C07141=1012.979,-24.500,-114.900,-28.755,51.503,-32.003
C07142=1012.980,-24.266,-114.919,-28.753,51.485,-32.004
C07143=1012.980,-24.032,-114.938,-28.751,51.466,-32.006
C07144=1012.980,-23.797,-114.958,-28.749,51.447,-32.007
C07145=1012.981,-23.564,-114.978,-28.747,51.429,-32.008
C07146=1012.981,-23.329,-114.997,-28.745,51.412,-32.007
C07147=1012.981,-23.095,-115.017,-28.743,51.394,-32.009
C07148=1012.982,-22.861,-115.036,-28.741,51.376,-32.010
C07149=1012.982,-22.628,-115.056,-28.739,51.359,-32.010
C07150=1012.982,-22.394,-115.076,-28.737,51.342,-32.011
C07151=1012.982,-22.159,-115.095,-28.736,51.326,-32.012
C07152=1012.983,-21.925,-115.114,-28.734,51.309,-32.012
C07153=1012.983,-21.691,-115.135,-28.732,51.292,-32.013
C07154=1012.983,-21.457,-115.154,-28.730,51.276,-32.014
C07155=1012.984,-21.223,-115.173,-28.728,51.261,-32.015
C07156=1012.983,-20.989,-115.193,-28.726,51.246,-32.014
C07157=1012.984,-20.755,-115.213,-28.725,51.230,-32.015
C07158=1012.985,-20.521,-115.232,-28.723,51.215,-32.015
C07159=1012.984,-20.243,-115.255,-28.721,51.197,-32.016
C07160=1012.985,-19.894,-115.285,-28.718,51.175,-32.016
C07161=1012.986,-19.633,-115.306,-28.717,51.160,-32.017
C07162=1012.986,-19.334,-115.331,-28.714,51.142,-32.017
C07163=1012.986,-19.008,-115.359,-28.712,51.123,-32.017
C07164=1012.987,-18.676,-115.386,-28.710,51.105,-32.018
C07165=1012.986,-18.359,-115.413,-28.708,51.087,-32.018
C07166=1012.987,-18.074,-115.437,-28.706,51.072,-32.017
C07167=1012.987,-17.827,-115.458,-28.704,51.058,-32.018
C07168=1012.987,-17.596,-115.477,-28.703,51.046,-32.018
C07169=1012.987,-17.366,-115.497,-28.702,51.035,-32.017
C07170=1012.988,-17.131,-115.516,-28.700,51.023,-32.017
C07171=1012.988,-16.894,-115.536,-28.699,51.011,-32.017
C07172=1012.987,-16.657,-115.556,-28.697,50.999,-32.017
C07173=1012.988,-16.421,-115.575,-28.696,50.989,-32.016
C07174=1012.988,-16.187,-115.595,-28.695,50.979,-32.016
C07175=1012.988,-15.950,-115.616,-28.693,50.967,-32.017
C07176=1012.989,-15.715,-115.634,-28.692,50.957,-32.016
C07177=1012.988,-15.481,-115.655,-28.691,50.947,-32.016
C07178=1012.989,-15.253,-115.673,-28.690,50.937,-32.016
C07179=1012.989,-15.025,-115.692,-28.688,50.928,-32.014
C07180=1012.989,-14.801,-115.712,-28.687,50.919,-32.013
C07181=1012.988,-14.578,-115.730,-28.686,50.909,-32.013
C07182=1012.989,-14.355,-115.749,-28.685,50.901,-32.012
C07183=1012.989,-14.131,-115.768,-28.683,50.893,-32.011
C07184=1012.989,-13.906,-115.786,-28.682,50.885,-32.009
C07185=1012.989,-13.676,-115.806,-28.681,50.878,-32.009
C07186=1012.989,-13.443,-115.825,-28.680,50.869,-32.008
C07187=1012.989,-13.206,-115.845,-28.679,50.861,-32.007
C07188=1012.989,-12.965,-115.865,-28.678,50.853,-32.007
C07189=1012.989,-12.720,-115.886,-28.677,50.846,-32.007
C07190=1012.990,-12.475,-115.906,-28.676,50.838,-32.006
C07191=1012.990,-12.228,-115.927,-28.675,50.831,-32.004
C07192=1012.989,-11.982,-115.948,-28.674,50.824,-32.003
C07193=1012.989,-11.734,-115.968,-28.673,50.817,-32.003
C07194=1012.989,-11.486,-115.990,-28.672,50.810,-32.001
C07195=1012.989,-11.237,-116.011,-28.671,50.804,-32.000
C07196=1012.989,-10.989,-116.031,-28.670,50.798,-31.999
C07197=1012.989,-10.739,-116.052,-28.669,50.793,-31.997
C07198=1012.989,-10.489,-116.073,-28.668,50.787,-31.996
C07199=1012.989,-10.239,-116.094,-28.667,50.782,-31.994
C07200=1012.990,-9.989,-116.115,-28.666,50.776,-31.993
C07201=1012.989,-9.738,-116.136,-28.666,50.772,-31.991
C07202=1012.989,-9.487,-116.157,-28.665,50.767,-31.989
C07203=1012.989,-9.236,-116.179,-28.664,50.763,-31.988
C07204=1012.989,-8.985,-116.199,-28.663,50.758,-31.986
C07205=1012.989,-8.733,-116.221,-28.662,50.754,-31.985
C07206=1012.989,-8.481,-116.242,-28.661,50.751,-31.982
C07207=1012.989,-8.230,-116.263,-28.661,50.748,-31.981
C07208=1012.989,-7.978,-116.284,-28.660,50.745,-31.979
C07209=1012.989,-7.724,-116.305,-28.659,50.742,-31.976
C07210=1012.989,-7.470,-116.327,-28.659,50.739,-31.975
C07211=1012.988,-7.215,-116.348,-28.658,50.737,-31.974
C07212=1012.988,-6.959,-116.369,-28.658,50.735,-31.970
C07213=1012.988,-6.702,-116.391,-28.657,50.734,-31.969
C07214=1012.987,-6.444,-116.413,-28.657,50.731,-31.967
C07215=1012.988,-6.186,-116.434,-28.656,50.730,-31.964
C07216=1012.987,-5.928,-116.456,-28.655,50.729,-31.961
C07217=1012.987,-5.670,-116.477,-28.655,50.728,-31.960
C07218=1012.987,-5.413,-116.499,-28.655,50.728,-31.957
C07219=1012.986,-5.161,-116.521,-28.654,50.728,-31.955
C07220=1012.987,-4.917,-116.541,-28.654,50.728,-31.953
C07221=1012.987,-4.682,-116.561,-28.654,50.728,-31.951
C07222=1012.986,-4.453,-116.580,-28.653,50.729,-31.948
C07223=1012.986,-4.227,-116.599,-28.653,50.729,-31.946
C07224=1012.986,-4.001,-116.618,-28.652,50.731,-31.943
C07225=1012.986,-3.771,-116.637,-28.652,50.731,-31.939
C07226=1012.986,-3.534,-116.658,-28.652,50.732,-31.938
C07227=1012.985,-3.292,-116.678,-28.651,50.734,-31.935
C07228=1012.985,-3.047,-116.698,-28.651,50.736,-31.933
C07229=1012.985,-2.802,-116.719,-28.651,50.738,-31.931
C07230=1012.985,-2.558,-116.739,-28.651,50.741,-31.926
C07231=1012.984,-2.315,-116.760,-28.651,50.743,-31.924
C07232=1012.984,-2.072,-116.781,-28.651,50.746,-31.922
C07233=1012.984,-1.830,-116.800,-28.650,50.749,-31.919
C07234=1012.983,-1.589,-116.821,-28.650,50.753,-31.915
C07235=1012.983,-1.348,-116.841,-28.650,50.755,-31.913
C07236=1012.983,-1.109,-116.861,-28.650,50.758,-31.910
C07237=1012.982,-0.869,-116.882,-28.650,50.763,-31.907
C07238=1012.983,-0.631,-116.902,-28.650,50.767,-31.905
C07239=1012.982,-0.393,-116.922,-28.650,50.772,-31.901
C07240=1012.982,-0.156,-116.941,-28.650,50.776,-31.898
C07241=1012.982,0.079,-116.961,-28.650,50.780,-31.895
C07242=1012.980,0.314,-116.981,-28.650,50.785,-31.891
C07243=1012.980,0.548,-117.001,-28.650,50.790,-31.889
C07244=1012.980,0.784,-117.021,-28.650,50.795,-31.885
C07245=1012.980,1.019,-117.040,-28.650,50.801,-31.882
C07246=1012.980,1.256,-117.060,-28.650,50.807,-31.878
C07247=1012.979,1.492,-117.080,-28.650,50.813,-31.875
C07248=1012.979,1.727,-117.100,-28.650,50.819,-31.872
C07249=1012.978,1.956,-117.119,-28.651,50.825,-31.868
C07250=1012.978,2.177,-117.138,-28.651,50.832,-31.866
C07251=1012.978,2.585,-117.172,-28.651,50.843,-31.859
C07252=1012.977,2.969,-117.205,-28.652,50.856,-31.853
C07253=1012.976,3.360,-117.238,-28.652,50.868,-31.847
C07254=1012.975,3.569,-117.255,-28.652,50.875,-31.844
C07255=1012.976,3.788,-117.273,-28.653,50.883,-31.840
C07256=1012.975,4.016,-117.293,-28.653,50.890,-31.836
C07257=1012.974,4.249,-117.312,-28.653,50.899,-31.833
C07258=1012.974,4.481,-117.332,-28.654,50.907,-31.829
C07259=1012.974,4.713,-117.351,-28.654,50.916,-31.825
C07260=1012.973,4.944,-117.371,-28.654,50.925,-31.822
C07261=1012.973,5.176,-117.390,-28.655,50.935,-31.818
C07262=1012.972,5.408,-117.410,-28.655,50.943,-31.814
C07263=1012.972,5.641,-117.430,-28.656,50.953,-31.810
C07264=1012.971,5.875,-117.449,-28.656,50.963,-31.806
C07265=1012.971,6.109,-117.469,-28.656,50.973,-31.802
C07266=1012.970,6.343,-117.488,-28.657,50.983,-31.798
C07267=1012.970,6.576,-117.509,-28.657,50.993,-31.794
C07268=1012.970,6.806,-117.528,-28.658,51.004,-31.789
C07269=1012.969,7.036,-117.547,-28.658,51.015,-31.786
C07270=1012.968,7.263,-117.566,-28.659,51.025,-31.782
C07271=1012.968,7.489,-117.585,-28.660,51.037,-31.777
C07272=1012.967,7.715,-117.604,-28.660,51.048,-31.774
C07273=1012.966,7.939,-117.623,-28.661,51.059,-31.769
C07274=1012.966,8.162,-117.642,-28.661,51.070,-31.765
C07275=1012.965,8.385,-117.661,-28.662,51.082,-31.761
C07276=1012.965,8.608,-117.680,-28.662,51.093,-31.756
C07277=1012.965,8.830,-117.698,-28.663,51.106,-31.752
C07278=1012.964,9.052,-117.718,-28.664,51.118,-31.748
C07279=1012.964,9.275,-117.737,-28.664,51.130,-31.744
C07280=1012.963,9.498,-117.755,-28.665,51.142,-31.739
C07281=1012.962,9.721,-117.774,-28.666,51.154,-31.735
C07282=1012.962,9.944,-117.792,-28.667,51.167,-31.731
C07283=1012.961,10.168,-117.812,-28.667,51.180,-31.726
C07284=1012.961,10.394,-117.830,-28.668,51.194,-31.723
C07285=1012.960,10.618,-117.850,-28.669,51.207,-31.718
C07286=1012.960,10.839,-117.868,-28.670,51.222,-31.713
C07287=1012.959,11.056,-117.886,-28.670,51.234,-31.709
C07288=1012.958,11.272,-117.905,-28.671,51.248,-31.704
C07289=1012.958,11.488,-117.922,-28.672,51.262,-31.699
C07290=1012.957,11.708,-117.942,-28.673,51.276,-31.695
C07291=1012.956,11.931,-117.960,-28.673,51.290,-31.690
C07292=1012.956,12.158,-117.980,-28.674,51.305,-31.686
C07293=1012.955,12.387,-117.999,-28.675,51.320,-31.681
C07294=1012.954,12.615,-118.018,-28.676,51.336,-31.677
C07295=1012.954,12.844,-118.038,-28.677,51.351,-31.672
C07296=1012.954,13.072,-118.057,-28.678,51.367,-31.666
C07297=1012.953,13.300,-118.076,-28.679,51.383,-31.661
C07298=1012.952,13.527,-118.095,-28.680,51.399,-31.656
C07299=1012.952,13.755,-118.114,-28.681,51.416,-31.651
C07300=1012.951,13.982,-118.133,-28.682,51.432,-31.646
C07301=1012.951,14.208,-118.153,-28.683,51.449,-31.642
C07302=1012.949,14.434,-118.172,-28.684,51.465,-31.637
C07303=1012.949,14.660,-118.191,-28.685,51.481,-31.632
C07304=1012.948,14.886,-118.209,-28.686,51.499,-31.626
C07305=1012.948,15.113,-118.229,-28.687,51.516,-31.622
C07306=1012.947,15.340,-118.248,-28.688,51.534,-31.617
C07307=1012.946,15.565,-118.267,-28.689,51.552,-31.611
C07308=1012.945,15.792,-118.287,-28.690,51.570,-31.606
C07309=1012.944,16.019,-118.305,-28.691,51.588,-31.600
C07310=1012.944,16.247,-118.325,-28.693,51.606,-31.595
C07311=1012.943,16.474,-118.344,-28.694,51.625,-31.590
C07312=1012.943,16.703,-118.364,-28.695,51.643,-31.585
C07313=1012.942,16.931,-118.383,-28.696,51.663,-31.579
C07314=1012.940,17.161,-118.402,-28.697,51.682,-31.574
C07315=1012.940,17.392,-118.421,-28.699,51.702,-31.568
C07316=1012.939,17.623,-118.441,-28.700,51.722,-31.562
C07317=1012.939,17.855,-118.460,-28.701,51.742,-31.557
C07318=1012.938,18.087,-118.480,-28.702,51.762,-31.551
C07319=1012.937,18.320,-118.500,-28.704,51.783,-31.546
C07320=1012.936,18.553,-118.520,-28.705,51.803,-31.540
C07321=1012.935,18.786,-118.539,-28.707,51.824,-31.535
C07322=1012.934,19.048,-118.562,-28.708,51.848,-31.529
C07323=1012.933,19.353,-118.587,-28.710,51.876,-31.521
C07324=1012.931,19.749,-118.621,-28.712,51.913,-31.511
C07325=1012.930,20.049,-118.647,-28.714,51.941,-31.504
C07326=1012.929,20.367,-118.673,-28.716,51.972,-31.495
C07327=1012.928,20.687,-118.700,-28.718,52.002,-31.488
C07328=1012.927,20.997,-118.726,-28.720,52.033,-31.479
C07329=1012.926,21.286,-118.751,-28.722,52.062,-31.472
C07330=1012.925,21.545,-118.773,-28.724,52.088,-31.465
C07331=1012.923,21.956,-118.807,-28.726,52.129,-31.455
C07332=1012.922,22.369,-118.842,-28.729,52.172,-31.443
C07333=1012.921,22.713,-118.871,-28.731,52.208,-31.435
C07334=1012.919,23.005,-118.896,-28.733,52.238,-31.427
C07335=1012.918,23.306,-118.922,-28.736,52.270,-31.419
C07336=1012.917,23.669,-118.953,-28.738,52.309,-31.409
C07337=1012.916,23.879,-118.970,-28.740,52.331,-31.404
C07338=1012.916,24.101,-118.989,-28.741,52.356,-31.397
C07339=1012.914,24.333,-119.009,-28.743,52.381,-31.392
C07340=1012.913,24.569,-119.029,-28.745,52.408,-31.386
C07341=1012.912,24.804,-119.048,-28.746,52.434,-31.379
C07342=1012.911,25.040,-119.068,-28.748,52.460,-31.373
C07343=1012.910,25.276,-119.088,-28.750,52.486,-31.366
C07344=1012.909,25.512,-119.108,-28.752,52.514,-31.361
C07345=1012.907,25.749,-119.128,-28.754,52.542,-31.353
C07346=1012.907,25.986,-119.149,-28.756,52.568,-31.347
C07347=1012.906,26.222,-119.168,-28.757,52.596,-31.340
C07348=1012.905,26.459,-119.189,-28.759,52.624,-31.334
C07349=1012.904,26.694,-119.208,-28.761,52.651,-31.327
C07350=1012.903,26.929,-119.228,-28.763,52.680,-31.320
C07351=1012.902,27.163,-119.248,-28.765,52.708,-31.313
C07352=1012.901,27.396,-119.268,-28.767,52.737,-31.307
C07353=1012.899,27.630,-119.288,-28.769,52.764,-31.301
C07354=1012.899,27.864,-119.307,-28.770,52.794,-31.293
C07355=1012.898,28.099,-119.327,-28.772,52.822,-31.287
C07356=1012.897,28.333,-119.347,-28.774,52.851,-31.281
C07357=1012.896,28.566,-119.367,-28.777,52.881,-31.275
C07358=1012.895,28.802,-119.386,-28.778,52.910,-31.267
C07359=1012.893,29.037,-119.406,-28.780,52.939,-31.261
C07360=1012.892,29.272,-119.427,-28.782,52.969,-31.254
C07361=1012.891,29.507,-119.446,-28.784,53.000,-31.247
C07362=1012.890,29.744,-119.466,-28.786,53.030,-31.240
C07363=1012.889,29.978,-119.487,-28.789,53.061,-31.233
C07364=1012.888,30.214,-119.506,-28.790,53.091,-31.226
C07365=1012.887,30.449,-119.526,-28.793,53.122,-31.219
C07366=1012.886,30.684,-119.547,-28.795,53.153,-31.213
C07367=1012.885,30.919,-119.566,-28.797,53.184,-31.206
C07368=1012.883,31.155,-119.586,-28.799,53.217,-31.199
C07369=1012.882,31.390,-119.606,-28.801,53.248,-31.193
C07370=1012.882,31.624,-119.626,-28.804,53.281,-31.186
C07371=1012.881,31.860,-119.645,-28.806,53.312,-31.178
C07372=1012.879,32.095,-119.665,-28.808,53.344,-31.172
C07373=1012.878,32.330,-119.685,-28.810,53.377,-31.165
C07374=1012.877,32.565,-119.705,-28.812,53.409,-31.158
C07375=1012.876,32.801,-119.725,-28.815,53.442,-31.151
C07376=1012.874,33.036,-119.745,-28.817,53.475,-31.145
C07377=1012.874,33.272,-119.765,-28.819,53.509,-31.136
C07378=1012.873,33.507,-119.785,-28.821,53.542,-31.130
C07379=1012.871,33.742,-119.805,-28.824,53.577,-31.122
C07380=1012.870,33.978,-119.825,-28.826,53.609,-31.115
C07381=1012.869,34.213,-119.845,-28.828,53.644,-31.108
C07382=1012.868,34.448,-119.865,-28.831,53.678,-31.102
C07383=1012.866,34.684,-119.885,-28.833,53.712,-31.094
C07384=1012.865,34.919,-119.905,-28.835,53.747,-31.088
C07385=1012.864,35.154,-119.925,-28.838,53.782,-31.080
C07386=1012.862,35.389,-119.945,-28.840,53.817,-31.073
C07387=1012.861,35.625,-119.965,-28.843,53.852,-31.066
C07388=1012.860,35.860,-119.984,-28.845,53.888,-31.058
C07389=1012.859,36.095,-120.005,-28.847,53.923,-31.051
C07390=1012.857,36.330,-120.024,-28.850,53.958,-31.045
C07391=1012.856,36.566,-120.044,-28.852,53.995,-31.037
C07392=1012.855,36.801,-120.064,-28.855,54.032,-31.030
C07393=1012.854,37.036,-120.084,-28.857,54.067,-31.023
C07394=1012.853,37.271,-120.104,-28.860,54.103,-31.016
C07395=1012.851,37.507,-120.124,-28.862,54.140,-31.008
C07396=1012.850,37.742,-120.143,-28.865,54.177,-31.001
C07397=1012.848,37.978,-120.164,-28.868,54.215,-30.994
C07398=1012.847,38.214,-120.184,-28.870,54.251,-30.987
C07399=1012.846,38.449,-120.204,-28.873,54.289,-30.980
C07400=1012.845,38.684,-120.224,-28.875,54.327,-30.972
C07401=1012.844,38.919,-120.244,-28.878,54.364,-30.965
C07402=1012.843,39.155,-120.263,-28.880,54.403,-30.957
C07403=1012.841,39.390,-120.283,-28.883,54.440,-30.951
C07404=1012.840,39.626,-120.303,-28.886,54.479,-30.943
C07405=1012.838,39.861,-120.324,-28.889,54.518,-30.936
C07406=1012.837,40.096,-120.343,-28.891,54.557,-30.928
C07407=1012.836,40.331,-120.363,-28.894,54.596,-30.921
C07408=1012.834,40.567,-120.383,-28.897,54.635,-30.914
C07409=1012.833,40.802,-120.403,-28.899,54.674,-30.906
C07410=1012.832,41.038,-120.422,-28.902,54.713,-30.899
C07411=1012.830,41.273,-120.443,-28.905,54.754,-30.892
C07412=1012.829,41.508,-120.463,-28.908,54.794,-30.885
C07413=1012.827,41.743,-120.483,-28.910,54.834,-30.876
C07414=1012.826,41.979,-120.502,-28.913,54.874,-30.870
C07415=1012.825,42.214,-120.522,-28.916,54.915,-30.863
C07416=1012.824,42.450,-120.542,-28.919,54.956,-30.855
C07417=1012.822,42.685,-120.562,-28.922,54.997,-30.847
C07418=1012.820,42.921,-120.582,-28.925,55.037,-30.840
C07419=1012.819,43.156,-120.602,-28.928,55.079,-30.833
C07420=1012.818,43.391,-120.622,-28.930,55.120,-30.826
C07421=1012.816,43.627,-120.642,-28.934,55.162,-30.819
C07422=1012.815,43.863,-120.662,-28.937,55.204,-30.812
C07423=1012.814,44.098,-120.682,-28.939,55.245,-30.803
C07424=1012.813,44.334,-120.702,-28.943,55.288,-30.797
C07425=1012.811,44.569,-120.722,-28.945,55.331,-30.789
C07426=1012.809,44.805,-120.742,-28.948,55.373,-30.781
C07427=1012.808,45.040,-120.762,-28.952,55.416,-30.775
C07428=1012.807,45.275,-120.781,-28.954,55.458,-30.767
C07429=1012.805,45.511,-120.802,-28.957,55.502,-30.760
C07430=1012.804,45.747,-120.821,-28.961,55.545,-30.753
C07431=1012.802,45.982,-120.841,-28.964,55.588,-30.746
C07432=1012.801,46.217,-120.861,-28.967,55.632,-30.739
C07433=1012.799,46.453,-120.881,-28.970,55.676,-30.730
C07434=1012.798,46.688,-120.901,-28.973,55.720,-30.724
C07435=1012.796,46.924,-120.920,-28.976,55.765,-30.715
C07436=1012.794,47.160,-120.941,-28.979,55.809,-30.709
C07437=1012.793,47.395,-120.960,-28.982,55.854,-30.701
C07438=1012.792,47.630,-120.980,-28.985,55.899,-30.694
C07439=1012.790,47.866,-121.000,-28.989,55.943,-30.687
C07440=1012.789,48.102,-121.021,-28.992,55.989,-30.680
C07441=1012.788,48.337,-121.041,-28.995,56.034,-30.673
C07442=1012.787,48.567,-121.060,-28.998,56.079,-30.665
C07443=1012.784,48.809,-121.080,-29.002,56.126,-30.657
C07444=1012.783,49.044,-121.100,-29.005,56.172,-30.650
C07445=1012.781,49.280,-121.120,-29.008,56.217,-30.644
C07446=1012.780,49.515,-121.140,-29.012,56.264,-30.636
C07447=1012.779,49.751,-121.160,-29.015,56.310,-30.629
C07448=1012.777,49.986,-121.180,-29.018,56.357,-30.622
C07449=1012.775,50.222,-121.200,-29.022,56.404,-30.614
C07450=1012.774,50.457,-121.219,-29.025,56.452,-30.606
C07451=1012.772,50.693,-121.240,-29.029,56.498,-30.600
C07452=1012.771,50.928,-121.259,-29.032,56.546,-30.593
C07453=1012.769,51.164,-121.279,-29.036,56.593,-30.586
C07454=1012.767,51.399,-121.300,-29.039,56.642,-30.578
C07455=1012.767,51.635,-121.320,-29.043,56.690,-30.571
C07456=1012.765,51.871,-121.340,-29.046,56.738,-30.564
C07457=1012.763,52.106,-121.360,-29.049,56.787,-30.557
C07458=1012.762,52.342,-121.379,-29.053,56.835,-30.550
C07459=1012.760,52.578,-121.400,-29.056,56.883,-30.542
C07460=1012.759,52.813,-121.419,-29.060,56.933,-30.536
C07461=1012.757,53.049,-121.440,-29.064,56.982,-30.529
C07462=1012.755,53.284,-121.459,-29.067,57.031,-30.521
C07463=1012.754,53.520,-121.478,-29.071,57.081,-30.515
C07464=1012.752,53.756,-121.499,-29.075,57.130,-30.507
C07465=1012.751,53.991,-121.518,-29.078,57.180,-30.500
C07466=1012.749,54.227,-121.539,-29.082,57.230,-30.494
C07467=1012.747,54.462,-121.558,-29.086,57.281,-30.486
C07468=1012.745,54.698,-121.579,-29.089,57.331,-30.479
C07469=1012.745,54.934,-121.599,-29.093,57.381,-30.473
C07470=1012.743,55.170,-121.619,-29.097,57.432,-30.466
C07471=1012.741,55.405,-121.639,-29.100,57.483,-30.458
C07472=1012.740,55.641,-121.658,-29.105,57.534,-30.452
C07473=1012.738,55.877,-121.678,-29.108,57.585,-30.445
C07474=1012.736,56.112,-121.698,-29.112,57.637,-30.438
C07475=1012.734,56.348,-121.718,-29.116,57.689,-30.431
C07476=1012.733,56.583,-121.738,-29.120,57.741,-30.425
C07477=1012.731,56.819,-121.758,-29.124,57.793,-30.418
C07478=1012.730,57.055,-121.778,-29.128,57.845,-30.412
C07479=1012.727,57.291,-121.797,-29.132,57.897,-30.403
C07480=1012.726,57.526,-121.817,-29.136,57.950,-30.397
C07481=1012.724,57.762,-121.837,-29.140,58.003,-30.390
C07482=1012.723,57.997,-121.857,-29.144,58.055,-30.384
C07483=1012.721,58.233,-121.877,-29.148,58.109,-30.377
C07484=1012.719,58.469,-121.897,-29.152,58.163,-30.370
C07485=1012.718,58.705,-121.918,-29.156,58.215,-30.364
C07486=1012.716,58.941,-121.937,-29.160,58.269,-30.358
C07487=1012.714,59.177,-121.957,-29.164,58.323,-30.352
C07488=1012.713,59.412,-121.977,-29.168,58.378,-30.344
C07489=1012.711,59.648,-121.997,-29.173,58.432,-30.338
C07490=1012.710,59.883,-122.017,-29.177,58.486,-30.331
C07491=1012.708,60.119,-122.037,-29.181,58.540,-30.325
C07492=1012.706,60.355,-122.056,-29.185,58.596,-30.318
C07493=1012.704,60.591,-122.077,-29.189,58.650,-30.312
C07494=1012.703,60.826,-122.096,-29.194,58.706,-30.305
C07495=1012.701,61.062,-122.117,-29.198,58.761,-30.299
C07496=1012.700,61.297,-122.136,-29.203,58.816,-30.294
C07497=1012.697,61.533,-122.156,-29.207,58.872,-30.287
C07498=1012.696,61.769,-122.176,-29.211,58.928,-30.281
C07499=1012.694,62.005,-122.196,-29.216,58.984,-30.275
C07500=1012.692,62.280,-122.219,-29.221,59.050,-30.267
C07501=1012.690,62.568,-122.243,-29.226,59.119,-30.259
C07502=1012.688,62.844,-122.266,-29.232,59.186,-30.252
C07503=1012.686,63.139,-122.292,-29.237,59.256,-30.246
C07504=1012.684,63.422,-122.315,-29.243,59.325,-30.237
C07505=1012.682,63.673,-122.336,-29.248,59.386,-30.231
C07506=1012.681,63.910,-122.356,-29.252,59.444,-30.225
C07507=1012.679,64.163,-122.378,-29.257,59.506,-30.219
C07508=1012.676,64.430,-122.401,-29.262,59.572,-30.212
C07509=1012.674,64.702,-122.423,-29.268,59.638,-30.206
C07510=1012.673,64.965,-122.445,-29.273,59.704,-30.199
C07511=1012.671,65.227,-122.467,-29.279,59.768,-30.193
C07512=1012.669,65.480,-122.489,-29.284,59.830,-30.187
C07513=1012.667,65.722,-122.509,-29.288,59.892,-30.180
C07514=1012.665,65.956,-122.529,-29.294,59.951,-30.176
C07515=1012.662,66.347,-122.562,-29.302,60.049,-30.166
C07516=1012.661,66.561,-122.580,-29.306,60.102,-30.161
C07517=1012.659,66.797,-122.599,-29.311,60.163,-30.156
C07518=1012.657,67.033,-122.619,-29.316,60.223,-30.150
C07519=1012.655,67.270,-122.639,-29.321,60.283,-30.145
C07520=1012.654,67.508,-122.659,-29.326,60.344,-30.140
C07521=1012.652,67.747,-122.680,-29.331,60.405,-30.133
C07522=1012.650,67.988,-122.700,-29.337,60.466,-30.129
C07523=1012.648,68.233,-122.721,-29.342,60.530,-30.123
C07524=1012.646,68.482,-122.741,-29.348,60.595,-30.118
C07525=1012.644,68.732,-122.763,-29.353,60.659,-30.114
C07526=1012.642,68.979,-122.784,-29.359,60.723,-30.108
C07527=1012.640,69.227,-122.804,-29.364,60.788,-30.103
C07528=1012.638,69.469,-122.825,-29.370,60.851,-30.097
C07529=1012.637,69.710,-122.845,-29.376,60.914,-30.093
C07530=1012.635,69.951,-122.866,-29.381,60.978,-30.088
C07531=1012.633,70.192,-122.885,-29.386,61.042,-30.082
C07532=1012.631,70.433,-122.906,-29.392,61.105,-30.078
C07533=1012.629,70.674,-122.926,-29.398,61.169,-30.074
C07534=1012.627,70.915,-122.946,-29.403,61.233,-30.068
C07535=1012.625,71.156,-122.967,-29.409,61.297,-30.064
C07536=1012.624,71.397,-122.987,-29.415,61.362,-30.060
C07537=1012.621,71.638,-123.007,-29.421,61.426,-30.055
C07538=1012.620,71.879,-123.027,-29.427,61.491,-30.051
C07539=1012.618,72.122,-123.048,-29.432,61.556,-30.046
C07540=1012.617,72.364,-123.068,-29.439,61.622,-30.042
C07541=1012.614,72.607,-123.089,-29.444,61.687,-30.037
C07542=1012.612,72.850,-123.109,-29.450,61.753,-30.032
C07543=1012.611,73.095,-123.130,-29.457,61.820,-30.029
C07544=1012.607,73.477,-123.162,-29.466,61.924,-30.022
C07545=1012.605,73.831,-123.191,-29.475,62.021,-30.016
C07546=1012.602,74.082,-123.213,-29.482,62.091,-30.012
C07547=1012.601,74.349,-123.236,-29.489,62.164,-30.008
C07548=1012.598,74.621,-123.258,-29.496,62.239,-30.005
C07549=1012.597,74.881,-123.280,-29.503,62.311,-30.001
C07550=1012.594,75.129,-123.301,-29.509,62.381,-29.997
C07551=1012.592,75.377,-123.322,-29.516,62.449,-29.993
C07552=1012.591,75.623,-123.342,-29.523,62.518,-29.990
C07553=1012.589,75.866,-123.362,-29.529,62.586,-29.987
C07554=1012.587,76.107,-123.383,-29.536,62.654,-29.982
C07555=1012.585,76.346,-123.403,-29.542,62.721,-29.980
C07556=1012.583,76.581,-123.422,-29.549,62.787,-29.976
C07557=1012.581,76.814,-123.442,-29.555,62.854,-29.974
C07558=1012.580,77.044,-123.461,-29.562,62.918,-29.971
C07559=1012.578,77.273,-123.481,-29.569,62.983,-29.969
C07560=1012.576,77.501,-123.500,-29.575,63.048,-29.965
C07561=1012.574,77.727,-123.519,-29.582,63.113,-29.963
C07562=1012.572,77.955,-123.538,-29.588,63.178,-29.961
C07563=1012.571,78.184,-123.557,-29.595,63.244,-29.958
C07564=1012.569,78.415,-123.576,-29.602,63.310,-29.956
C07565=1012.567,78.646,-123.596,-29.609,63.377,-29.954
C07566=1012.564,78.881,-123.616,-29.615,63.445,-29.951
C07567=1012.563,79.118,-123.636,-29.622,63.513,-29.948
C07568=1012.561,79.358,-123.656,-29.630,63.582,-29.947
C07569=1012.559,79.600,-123.677,-29.638,63.653,-29.946
C07570=1012.558,79.845,-123.696,-29.645,63.724,-29.944
C07571=1012.556,80.091,-123.717,-29.653,63.795,-29.941
C07572=1012.553,80.334,-123.737,-29.660,63.866,-29.940
C07573=1012.552,80.563,-123.757,-29.668,63.934,-29.938
C07574=1012.550,80.780,-123.775,-29.674,63.999,-29.936
C07575=1012.548,80.997,-123.793,-29.681,64.061,-29.935
C07576=1012.547,81.226,-123.812,-29.689,64.129,-29.934
C07577=1012.544,81.468,-123.833,-29.697,64.201,-29.934
C07578=1012.542,81.715,-123.854,-29.705,64.274,-29.931
C07579=1012.540,81.962,-123.874,-29.713,64.347,-29.931
C07580=1012.538,82.209,-123.895,-29.721,64.421,-29.929
C07581=1012.537,82.455,-123.915,-29.730,64.494,-29.929
C07582=1012.534,82.701,-123.936,-29.738,64.568,-29.928
C07583=1012.533,82.947,-123.957,-29.747,64.641,-29.928
C07584=1012.530,83.192,-123.977,-29.755,64.715,-29.927
C07585=1012.529,83.437,-123.998,-29.763,64.789,-29.925
C07586=1012.526,83.681,-124.018,-29.772,64.862,-29.926
C07587=1012.524,83.925,-124.038,-29.781,64.936,-29.925
C07588=1012.523,84.169,-124.059,-29.790,65.011,-29.925
C07589=1012.521,84.412,-124.079,-29.799,65.084,-29.926
C07590=1012.519,84.655,-124.099,-29.807,65.158,-29.925
C07591=1012.517,84.897,-124.119,-29.816,65.232,-29.925
C07592=1012.515,85.138,-124.140,-29.825,65.306,-29.925
C07593=1012.513,85.380,-124.160,-29.834,65.379,-29.927
C07594=1012.511,85.620,-124.180,-29.843,65.453,-29.926
C07595=1012.509,85.861,-124.200,-29.853,65.528,-29.927
C07596=1012.507,86.100,-124.220,-29.862,65.601,-29.929
C07597=1012.505,86.339,-124.240,-29.871,65.675,-29.929
C07598=1012.503,86.579,-124.260,-29.880,65.749,-29.930
C07599=1012.501,86.818,-124.280,-29.890,65.824,-29.932
C07600=1012.500,87.055,-124.300,-29.900,65.897,-29.934
C07601=1012.497,87.291,-124.320,-29.909,65.970,-29.934
C07602=1012.496,87.526,-124.340,-29.919,66.043,-29.937
C07603=1012.494,87.756,-124.358,-29.928,66.115,-29.938
C07604=1012.492,87.983,-124.378,-29.938,66.186,-29.941
C07605=1012.490,88.207,-124.397,-29.947,66.258,-29.941
C07606=1012.488,88.431,-124.415,-29.956,66.328,-29.943
C07607=1012.487,88.655,-124.434,-29.966,66.399,-29.945
C07608=1012.485,88.880,-124.453,-29.975,66.469,-29.947
C07609=1012.483,89.107,-124.472,-29.985,66.541,-29.949
C07610=1012.481,89.336,-124.490,-29.995,66.614,-29.952
C07611=1012.479,89.569,-124.511,-30.006,66.686,-29.956
C07612=1012.477,89.806,-124.530,-30.016,66.762,-29.958
C07613=1012.475,90.089,-124.554,-30.029,66.852,-29.961
C07614=1012.472,90.423,-124.582,-30.044,66.959,-29.966
C07615=1012.469,90.742,-124.609,-30.059,67.061,-29.971
C07616=1012.468,91.002,-124.630,-30.071,67.144,-29.975
C07617=1012.466,91.237,-124.649,-30.082,67.220,-29.978
C07618=1012.464,91.473,-124.669,-30.093,67.296,-29.981
C07619=1012.462,91.707,-124.689,-30.104,67.372,-29.985
C07620=1012.460,91.943,-124.708,-30.116,67.448,-29.990
C07621=1012.458,92.179,-124.729,-30.128,67.523,-29.995
C07622=1012.456,92.414,-124.747,-30.139,67.601,-29.999
C07623=1012.454,92.767,-124.777,-30.157,67.715,-30.006
C07624=1012.451,93.120,-124.807,-30.175,67.830,-30.014
C07625=1012.448,93.355,-124.827,-30.188,67.907,-30.020
C07626=1012.447,93.590,-124.846,-30.200,67.984,-30.024
C07627=1012.445,93.825,-124.865,-30.212,68.061,-30.030
C07628=1012.443,94.061,-124.885,-30.224,68.138,-30.035
C07629=1012.441,94.296,-124.905,-30.237,68.216,-30.041
C07630=1012.440,94.531,-124.924,-30.250,68.293,-30.047
C07631=1012.437,94.766,-124.944,-30.263,68.371,-30.053
C07632=1012.436,95.002,-124.964,-30.276,68.449,-30.060
C07633=1012.434,95.237,-124.983,-30.289,68.527,-30.066
C07634=1012.432,95.473,-125.003,-30.303,68.605,-30.073
C07635=1012.430,95.707,-125.022,-30.316,68.683,-30.080
C07636=1012.428,95.943,-125.042,-30.330,68.761,-30.087
C07637=1012.426,96.178,-125.062,-30.344,68.839,-30.095
C07638=1012.424,96.413,-125.082,-30.358,68.918,-30.103
C07639=1012.422,96.648,-125.100,-30.372,68.997,-30.109
C07640=1012.420,96.884,-125.121,-30.386,69.076,-30.118
C07641=1012.418,97.119,-125.140,-30.401,69.156,-30.126
C07642=1012.417,97.354,-125.160,-30.416,69.234,-30.136
C07643=1012.414,97.589,-125.180,-30.430,69.314,-30.144
C07644=1012.413,97.824,-125.199,-30.445,69.393,-30.152
C07645=1012.411,98.060,-125.218,-30.460,69.472,-30.162
C07646=1012.410,98.295,-125.238,-30.475,69.552,-30.171
C07647=1012.407,98.530,-125.258,-30.490,69.631,-30.179
C07648=1012.406,98.766,-125.277,-30.506,69.711,-30.190
C07649=1012.404,99.000,-125.297,-30.522,69.792,-30.200
C07650=1012.402,99.236,-125.317,-30.538,69.871,-30.210
C07651=1012.400,99.471,-125.336,-30.553,69.952,-30.219
C07652=1012.398,99.707,-125.355,-30.570,70.032,-30.230
C07653=1012.396,99.941,-125.375,-30.587,70.113,-30.242
C07654=1012.394,100.176,-125.395,-30.603,70.194,-30.251
C07655=1012.393,100.412,-125.414,-30.621,70.274,-30.265
C07656=1012.391,100.646,-125.434,-30.637,70.355,-30.275
C07657=1012.389,100.882,-125.453,-30.655,70.437,-30.287
C07658=1012.386,101.117,-125.473,-30.672,70.517,-30.299
C07659=1012.385,101.353,-125.492,-30.690,70.599,-30.312
C07660=1012.383,101.588,-125.512,-30.708,70.681,-30.325
C07661=1012.382,101.823,-125.531,-30.726,70.762,-30.337
C07662=1012.379,102.058,-125.551,-30.744,70.843,-30.349
C07663=1012.378,102.293,-125.571,-30.763,70.925,-30.364
C07664=1012.376,102.528,-125.590,-30.782,71.007,-30.378
C07665=1012.375,102.763,-125.610,-30.800,71.089,-30.390
C07666=1012.372,102.999,-125.629,-30.820,71.172,-30.406
C07667=1012.370,103.234,-125.649,-30.839,71.253,-30.420
C07668=1012.369,103.469,-125.668,-30.859,71.336,-30.434
C07669=1012.367,103.704,-125.688,-30.879,71.419,-30.451
C07670=1012.366,103.939,-125.707,-30.898,71.501,-30.464
C07671=1012.363,104.174,-125.727,-30.919,71.584,-30.480
C07672=1012.362,104.410,-125.747,-30.940,71.666,-30.497
C07673=1012.360,104.645,-125.766,-30.961,71.750,-30.514
C07674=1012.358,104.880,-125.785,-30.982,71.833,-30.530
C07675=1012.356,105.115,-125.805,-31.003,71.916,-30.547
C07676=1012.354,105.351,-125.825,-31.026,72.000,-30.565
C07677=1012.352,105.585,-125.844,-31.047,72.082,-30.582
C07678=1012.351,105.820,-125.864,-31.070,72.166,-30.601
C07679=1012.349,106.055,-125.883,-31.092,72.251,-30.618
C07680=1012.347,106.290,-125.903,-31.116,72.334,-30.638
C07681=1012.345,106.526,-125.922,-31.138,72.419,-30.656
C07682=1012.343,106.761,-125.942,-31.162,72.502,-30.676
C07683=1012.342,106.997,-125.961,-31.186,72.587,-30.695
C07684=1012.340,107.231,-125.981,-31.210,72.670,-30.715
C07685=1012.339,107.467,-126.001,-31.235,72.755,-30.736
C07686=1012.336,107.702,-126.020,-31.259,72.840,-30.756
C07687=1012.335,107.937,-126.040,-31.284,72.925,-30.778
C07688=1012.333,108.172,-126.060,-31.309,73.009,-30.798
C07689=1012.331,108.407,-126.078,-31.335,73.094,-30.821
C07690=1012.329,108.642,-126.098,-31.361,73.179,-30.844
C07691=1012.328,108.877,-126.117,-31.388,73.264,-30.867
C07692=1012.326,109.112,-126.137,-31.415,73.349,-30.890
C07693=1012.324,109.340,-126.156,-31.442,73.432,-30.915
C07694=1012.322,109.583,-126.177,-31.470,73.520,-30.939
C07695=1012.320,109.818,-126.196,-31.498,73.605,-30.963
C07696=1012.319,110.053,-126.216,-31.526,73.692,-30.988
C07697=1012.317,110.288,-126.234,-31.555,73.776,-31.014
C07698=1012.316,110.524,-126.254,-31.584,73.863,-31.040
C07699=1012.314,110.758,-126.273,-31.614,73.949,-31.066
C07700=1012.312,110.994,-126.294,-31.645,74.035,-31.095
C07701=1012.310,111.229,-126.313,-31.674,74.120,-31.121
C07702=1012.308,111.463,-126.332,-31.705,74.206,-31.148
C07703=1012.307,111.699,-126.352,-31.737,74.293,-31.178
C07704=1012.305,111.934,-126.371,-31.769,74.380,-31.207
C07705=1012.304,112.169,-126.391,-31.801,74.466,-31.236
C07706=1012.301,112.404,-126.410,-31.833,74.552,-31.266
C07707=1012.300,112.640,-126.429,-31.867,74.639,-31.298
C07708=1012.298,112.874,-126.449,-31.900,74.726,-31.327
C07709=1012.297,113.110,-126.468,-31.935,74.813,-31.360
C07710=1012.294,113.345,-126.488,-31.969,74.899,-31.391
C07711=1012.293,113.580,-126.508,-32.004,74.986,-31.424
C07712=1012.291,113.815,-126.527,-32.040,75.073,-31.458
C07713=1012.290,114.050,-126.547,-32.076,75.160,-31.492
C07714=1012.288,114.285,-126.567,-32.113,75.248,-31.526
C07715=1012.287,114.520,-126.586,-32.150,75.335,-31.562
C07716=1012.284,114.756,-126.605,-32.188,75.422,-31.597
C07717=1012.283,114.991,-126.625,-32.226,75.509,-31.633
C07718=1012.281,115.226,-126.644,-32.264,75.597,-31.669
C07719=1012.280,115.461,-126.664,-32.305,75.685,-31.708
C07720=1012.278,115.696,-126.683,-32.345,75.772,-31.746
C07721=1012.277,115.931,-126.703,-32.386,75.860,-31.786
C07722=1012.275,116.166,-126.722,-32.427,75.947,-31.825
C07723=1012.274,116.401,-126.742,-32.469,76.036,-31.865
C07724=1012.272,116.636,-126.761,-32.512,76.124,-31.907
C07725=1012.269,116.872,-126.781,-32.556,76.212,-31.950
C07726=1012.268,117.107,-126.800,-32.600,76.301,-31.992
C07727=1012.266,117.342,-126.820,-32.645,76.389,-32.036
C07728=1012.265,117.578,-126.839,-32.690,76.477,-32.079
C07729=1012.263,117.812,-126.859,-32.737,76.565,-32.125
C07730=1012.262,118.048,-126.879,-32.783,76.653,-32.170
C07731=1012.260,118.282,-126.898,-32.831,76.742,-32.216
C07732=1012.259,118.518,-126.918,-32.880,76.831,-32.264
C07733=1012.257,118.753,-126.937,-32.930,76.919,-32.313
C07734=1012.255,118.988,-126.957,-32.980,77.008,-32.364
C07735=1012.254,119.223,-126.976,-33.031,77.096,-32.413
C07736=1012.252,119.459,-126.995,-33.083,77.185,-32.465
C07737=1012.250,119.693,-127.014,-33.136,77.275,-32.516
C07738=1012.249,119.929,-127.034,-33.190,77.364,-32.570
C07739=1012.248,120.164,-127.054,-33.245,77.453,-32.624
C07740=1012.246,120.399,-127.073,-33.301,77.542,-32.680
C07741=1012.244,120.634,-127.093,-33.357,77.632,-32.735
C07742=1012.242,120.869,-127.112,-33.412,77.717,-32.790
C07743=1012.241,121.104,-127.132,-33.466,77.799,-32.844
C07744=1012.240,121.340,-127.152,-33.519,77.881,-32.896
C07745=1012.239,121.574,-127.172,-33.575,77.963,-32.951
C07746=1012.237,121.809,-127.191,-33.632,78.045,-33.009
C07747=1012.236,122.044,-127.211,-33.690,78.127,-33.067
C07748=1012.234,122.280,-127.231,-33.746,78.209,-33.122
C07749=1012.232,122.516,-127.251,-33.807,78.292,-33.184
C07750=1012.231,122.750,-127.271,-33.867,78.374,-33.244
C07751=1012.230,122.985,-127.291,-33.927,78.457,-33.303
C07752=1012.228,123.220,-127.311,-33.989,78.539,-33.366
C07753=1012.227,123.456,-127.330,-34.052,78.621,-33.429
C07754=1012.225,123.691,-127.350,-34.117,78.705,-33.494
C07755=1012.224,123.925,-127.370,-34.182,78.787,-33.560
C07756=1012.223,124.161,-127.390,-34.249,78.871,-33.627
C07757=1012.221,124.396,-127.410,-34.317,78.953,-33.695
C07758=1012.220,124.632,-127.430,-34.386,79.036,-33.765
C07759=1012.218,124.866,-127.450,-34.458,79.119,-33.837
C07760=1012.216,125.196,-127.477,-34.558,79.236,-33.938
C07761=1012.214,125.572,-127.509,-34.677,79.369,-34.058
C07762=1012.213,125.807,-127.529,-34.752,79.452,-34.134
C07763=1012.211,126.041,-127.549,-34.829,79.535,-34.212
C07764=1012.210,126.277,-127.568,-34.907,79.618,-34.291
C07765=1012.209,126.512,-127.588,-34.987,79.701,-34.372
C07766=1012.207,126.748,-127.608,-35.069,79.786,-34.454
C07767=1012.205,126.983,-127.628,-35.152,79.869,-34.538
C07768=1012.204,127.217,-127.648,-35.238,79.953,-34.626
C07769=1012.203,127.453,-127.668,-35.322,80.036,-34.711
C07770=1012.201,127.688,-127.688,-35.412,80.120,-34.802
C07771=1012.200,127.924,-127.707,-35.502,80.204,-34.893
C07772=1012.199,128.159,-127.727,-35.593,80.289,-34.986
C07773=1012.198,128.394,-127.748,-35.688,80.372,-35.083
C07774=1012.196,128.629,-127.767,-35.783,80.456,-35.179
C07775=1012.195,128.864,-127.787,-35.880,80.540,-35.278
C07776=1012.193,129.099,-127.806,-35.979,80.624,-35.378
C07777=1012.192,129.335,-127.826,-36.080,80.708,-35.481
C07778=1012.191,129.569,-127.846,-36.183,80.792,-35.585
C07779=1012.190,129.805,-127.866,-36.291,80.877,-35.695
C07780=1012.188,130.040,-127.886,-36.398,80.961,-35.804
C07781=1012.187,130.276,-127.906,-36.507,81.044,-35.915
C07782=1012.186,130.510,-127.926,-36.620,81.130,-36.030
C07783=1012.185,130.746,-127.946,-36.737,81.214,-36.149
C07784=1012.184,130.981,-127.965,-36.852,81.298,-36.265
C07785=1012.181,131.216,-127.985,-36.973,81.382,-36.389
C07786=1012.180,131.452,-128.005,-37.096,81.467,-36.514
C07787=1012.179,131.686,-128.025,-37.222,81.552,-36.642
C07788=1012.177,131.922,-128.045,-37.351,81.636,-36.774
C07789=1012.176,132.157,-128.065,-37.482,81.721,-36.908
C07790=1012.175,132.393,-128.085,-37.616,81.805,-37.044
C07791=1012.174,132.628,-128.104,-37.753,81.890,-37.183
C07792=1012.173,132.863,-128.125,-37.896,81.975,-37.329
C07793=1012.171,133.098,-128.144,-38.039,82.060,-37.475
C07794=1012.170,133.333,-128.164,-38.186,82.144,-37.624
C07795=1012.169,133.569,-128.184,-38.338,82.230,-37.779
C07796=1012.167,133.804,-128.204,-38.491,82.314,-37.935
C07797=1012.166,134.039,-128.224,-38.651,82.399,-38.097
C07798=1012.165,134.274,-128.244,-38.815,82.484,-38.264
C07799=1012.164,134.510,-128.263,-38.980,82.568,-38.432
C07800=1012.163,134.749,-128.283,-39.153,82.655,-38.608
C07801=1012.161,135.045,-128.309,-39.374,82.762,-38.833
C07802=1012.160,135.330,-128.333,-39.595,82.864,-39.059
C07803=1012.159,135.564,-128.352,-39.782,82.949,-39.249
C07804=1012.158,135.788,-128.371,-39.964,83.030,-39.434
C07805=1012.156,136.207,-128.407,-40.319,83.180,-39.796
C07806=1012.153,136.593,-128.439,-40.661,83.320,-40.143
C07807=1012.151,136.977,-128.472,-41.015,83.457,-40.502
C07808=1012.149,137.394,-128.507,-41.420,83.608,-40.914
C07809=1012.147,137.777,-128.539,-41.813,83.745,-41.313
C07810=1012.146,138.198,-128.575,-42.261,83.897,-41.768
C07811=1012.145,138.450,-128.596,-42.544,83.987,-42.056
C07812=1012.143,138.724,-128.620,-42.861,84.085,-42.378
C07813=1012.142,139.018,-128.644,-43.210,84.190,-42.732
C07814=1012.140,139.326,-128.670,-43.594,84.300,-43.122
C07815=1012.139,139.639,-128.697,-44.004,84.412,-43.538
C07816=1012.137,139.947,-128.723,-44.421,84.522,-43.961
C07817=1012.136,140.243,-128.748,-44.835,84.627,-44.380
C07818=1012.135,140.518,-128.771,-45.241,84.725,-44.790
C07819=1012.134,140.902,-128.804,-45.837,84.861,-45.395
C07820=1012.132,141.077,-128.818,-46.116,84.923,-45.677
C07821=1012.132,141.327,-128.840,-46.531,85.011,-46.097
C07822=1012.131,141.529,-128.857,-46.876,85.082,-46.446
C07823=1012.130,141.774,-128.877,-47.312,85.168,-46.888
C07824=1012.128,142.014,-128.898,-47.752,85.252,-47.333
C07825=1012.127,142.252,-128.918,-48.208,85.336,-47.794
C07826=1012.127,142.491,-128.938,-48.681,85.419,-48.272
C07827=1012.125,142.732,-128.958,-49.171,85.502,-48.767
C07828=1012.124,142.971,-128.978,-49.681,85.584,-49.282
C07829=1012.123,143.211,-128.999,-50.217,85.667,-49.825
C07830=1012.122,143.452,-129.020,-50.776,85.750,-50.388
C07831=1012.122,143.692,-129.040,-51.356,85.832,-50.975
C07832=1012.121,143.933,-129.060,-51.961,85.914,-51.585
C07833=1012.119,144.173,-129.080,-52.591,85.996,-52.220
C07834=1012.119,144.415,-129.101,-53.247,86.077,-52.882
C07835=1012.118,144.656,-129.122,-53.932,86.157,-53.572
C07836=1012.117,144.897,-129.142,-54.655,86.238,-54.302
C07837=1012.115,145.140,-129.162,-55.400,86.317,-55.053
C07838=1012.114,145.381,-129.183,-56.188,86.396,-55.848
C07839=1012.114,145.623,-129.204,-57.014,86.475,-56.680
C07840=1012.113,145.865,-129.224,-57.865,86.552,-57.537
C07841=1012.112,146.107,-129.245,-58.769,86.629,-58.447
C07842=1012.111,146.349,-129.265,-59.716,86.705,-59.400
C07843=1012.110,146.592,-129.285,-60.707,86.781,-60.397
C07844=1012.109,146.834,-129.306,-61.746,86.855,-61.442
C07845=1012.108,147.078,-129.327,-62.847,86.929,-62.551
C07846=1012.108,147.326,-129.347,-64.020,87.002,-63.731
C07847=1012.107,147.580,-129.369,-65.276,87.076,-64.994
C07848=1012.105,147.842,-129.392,-66.645,87.151,-66.370
C07849=1012.105,148.112,-129.414,-68.149,87.227,-67.882
C07850=1012.103,148.390,-129.438,-69.775,87.302,-69.516
C07851=1012.102,148.675,-129.462,-71.541,87.378,-71.290
C07852=1012.101,148.967,-129.487,-73.451,87.452,-73.209
C07853=1012.100,149.264,-129.512,-75.517,87.524,-75.284
C07854=1012.099,149.562,-129.537,-77.725,87.594,-77.500
C07855=1012.099,149.863,-129.563,-80.068,87.659,-79.852
C07856=1012.098,150.162,-129.588,-82.536,87.721,-82.329
C07857=1012.096,150.460,-129.614,-85.121,87.778,-84.923
C07858=1012.096,150.752,-129.639,-87.799,87.829,-87.611
C07859=1012.095,151.038,-129.663,-90.525,87.873,-90.347
C07860=1012.094,151.318,-129.687,-93.298,87.913,-93.128
C07861=1012.093,151.588,-129.709,-96.091,87.946,-95.930
C07862=1012.092,151.851,-129.732,-98.883,87.973,-98.730
C07863=1012.091,152.106,-129.753,-101.679,87.995,-101.535
C07864=1012.091,152.354,-129.774,-104.442,88.012,-104.307
C07865=1012.090,152.598,-129.795,-107.179,88.023,-107.051
///RCONF 0,0,0,0,0,0,0,0,0,0,0,0,0,0,0,0,0,0,0,0,0,0,0,0
C07866=1012.090,152.841,-129.816,-109.917,88.030,-109.798
C07867=1012.089,153.083,-129.836,-112.710,88.032,-112.600
C07868=1012.088,153.324,-129.857,-115.482,88.030,-115.380
C07869=1012.088,153.565,-129.877,-118.239,88.023,-118.145
C07870=1012.087,153.807,-129.898,-120.969,88.011,-120.883
C07871=1012.086,154.048,-129.918,-123.660,87.995,-123.583
C07872=1012.085,154.289,-129.939,-126.301,87.975,-126.232
C07873=1012.085,154.530,-129.960,-128.881,87.950,-128.821
C07874=1012.084,154.770,-129.980,-131.394,87.921,-131.343
C07875=1012.084,155.011,-130.001,-133.831,87.888,-133.789
C07876=1012.083,155.252,-130.021,-136.188,87.852,-136.155
C07877=1012.081,155.616,-130.052,-139.638,87.789,-139.617
C07878=1012.081,155.971,-130.082,-142.768,87.722,-142.761
C07879=1012.080,156.209,-130.103,-144.776,87.672,-144.779
C07880=1012.080,156.449,-130.123,-146.697,87.620,-146.709
C07881=1012.079,156.688,-130.143,-148.553,87.565,-148.574
C07882=1012.079,156.928,-130.163,-150.302,87.508,-150.332
C07883=1012.078,157.167,-130.184,-151.997,87.447,-152.037
C07884=1012.078,157.407,-130.205,-153.604,87.385,-153.653
C07885=1012.078,157.645,-130.225,-155.114,87.322,-155.173
C07886=1012.077,157.882,-130.245,-156.570,87.256,-156.638
C07887=1012.076,158.120,-130.265,-157.932,87.190,-158.010
C07888=1012.076,158.356,-130.285,-159.251,87.121,-159.339
C07889=1012.075,158.592,-130.305,-160.485,87.051,-160.582
C07890=1012.075,158.828,-130.326,-161.660,86.980,-161.767
C07891=1012.074,159.063,-130.345,-162.799,86.907,-162.916
C07892=1012.074,159.299,-130.366,-163.880,86.834,-164.006
C07893=1012.073,159.535,-130.386,-164.898,86.759,-165.035
C07894=1012.073,159.769,-130.406,-165.881,86.684,-166.027
C07895=1012.072,160.002,-130.426,-166.804,86.608,-166.960
C07896=1012.071,160.234,-130.448,-167.215,86.573,-167.375
C07897=1012.071,160.468,-130.472,-167.299,86.565,-167.462
C07898=1012.070,160.709,-130.497,-167.381,86.557,-167.545
C07899=1012.070,160.959,-130.522,-167.478,86.549,-167.644
C07900=1012.069,161.221,-130.550,-167.564,86.540,-167.731
C07901=1012.069,161.498,-130.579,-167.675,86.530,-167.844
C07902=1012.068,161.791,-130.609,-167.773,86.520,-167.944
C07903=1012.067,162.095,-130.640,-167.870,86.511,-168.042
C07904=1012.066,162.401,-130.671,-167.981,86.500,-168.156
C07905=1012.065,162.692,-130.702,-168.077,86.491,-168.254
C07906=1012.064,163.000,-130.734,-168.187,86.480,-168.366
C07907=1012.063,163.294,-130.764,-168.282,86.471,-168.462
C07908=1012.063,163.558,-130.791,-168.374,86.462,-168.556
C07909=1012.062,163.795,-130.816,-168.453,86.454,-168.637
C07910=1012.061,164.016,-130.839,-168.530,86.446,-168.715
C07911=1012.060,164.350,-130.874,-168.638,86.436,-168.824
C07912=1012.059,164.624,-130.902,-168.730,86.426,-168.918
C07913=1012.059,164.942,-130.935,-168.836,86.415,-169.026
C07914=1012.058,165.245,-130.966,-168.927,86.406,-169.119
C07915=1012.057,165.481,-130.990,-169.003,86.398,-169.198
C07916=1012.057,165.716,-131.015,-169.090,86.389,-169.285
C07917=1012.057,165.953,-131.039,-169.166,86.381,-169.363
C07918=1012.056,166.188,-131.064,-169.227,86.374,-169.426
C07919=1012.055,166.423,-131.088,-169.301,86.366,-169.501
C07920=1012.055,166.658,-131.112,-169.375,86.358,-169.577
C07921=1012.054,166.895,-131.137,-169.448,86.350,-169.651
C07922=1012.054,167.130,-131.162,-169.534,86.342,-169.739
C07923=1012.052,167.366,-131.186,-169.608,86.333,-169.814
C07924=1012.052,167.601,-131.211,-169.680,86.326,-169.887
C07925=1012.052,167.837,-131.235,-169.752,86.317,-169.962
C07926=1012.050,168.073,-131.259,-169.837,86.308,-170.048
C07927=1012.050,168.308,-131.284,-169.908,86.301,-170.120
C07928=1012.049,168.544,-131.308,-169.980,86.292,-170.194
C07929=1012.049,168.779,-131.333,-170.050,86.285,-170.265
C07930=1012.048,169.015,-131.357,-170.121,86.276,-170.338
C07931=1012.048,169.251,-131.382,-170.191,86.269,-170.409
C07932=1012.047,169.486,-131.406,-170.261,86.260,-170.482
C07933=1012.047,169.722,-131.431,-170.331,86.252,-170.554
C07934=1012.046,169.958,-131.455,-170.413,86.243,-170.637
C07935=1012.045,170.193,-131.480,-170.482,86.234,-170.708
C07936=1012.045,170.429,-131.504,-170.552,86.226,-170.779
C07937=1012.045,170.664,-131.529,-170.619,86.218,-170.848
C07938=1012.044,170.900,-131.554,-170.688,86.210,-170.919
C07939=1012.043,171.136,-131.578,-170.755,86.202,-170.987
C07940=1012.042,171.371,-131.603,-170.823,86.194,-171.057
C07941=1012.042,171.607,-131.627,-170.902,86.185,-171.137
C07942=1012.041,171.843,-131.652,-170.968,86.177,-171.205
C07943=1012.041,172.079,-131.677,-171.035,86.169,-171.273
C07944=1012.040,172.314,-131.702,-171.113,86.160,-171.353
C07945=1012.040,172.550,-131.725,-171.179,86.151,-171.421
C07946=1012.039,172.786,-131.751,-171.245,86.143,-171.489
C07947=1012.038,173.021,-131.775,-171.311,86.134,-171.557
C07948=1012.038,173.257,-131.800,-171.375,86.126,-171.622
C07949=1012.037,173.493,-131.824,-171.440,86.118,-171.689
C07950=1012.037,173.729,-131.849,-171.505,86.109,-171.756
C07951=1012.036,173.964,-131.873,-171.581,86.100,-171.833
C07952=1012.036,174.200,-131.899,-171.645,86.092,-171.899
C07953=1012.035,174.435,-131.923,-171.709,86.083,-171.965
C07954=1012.035,174.672,-131.948,-171.784,86.074,-172.041
C07955=1012.034,174.907,-131.972,-171.847,86.066,-172.106
C07956=1012.033,175.143,-131.997,-171.910,86.057,-172.171
C07957=1012.033,175.378,-132.022,-171.972,86.049,-172.236
C07958=1012.032,175.615,-132.046,-172.034,86.041,-172.299
C07959=1012.032,175.850,-132.071,-172.107,86.032,-172.373
C07960=1012.032,176.086,-132.096,-172.169,86.023,-172.437
C07961=1012.031,176.321,-132.120,-172.230,86.015,-172.500
C07962=1012.030,176.557,-132.145,-172.292,86.006,-172.564
C07963=1012.030,176.794,-132.170,-172.364,85.997,-172.637
C07964=1012.029,177.029,-132.195,-172.424,85.988,-172.699
C07965=1012.030,177.265,-132.220,-172.495,85.979,-172.772
C07966=1012.028,177.501,-132.244,-172.556,85.970,-172.835
C07967=1012.028,177.736,-132.269,-172.615,85.962,-172.896
C07968=1012.027,177.972,-132.293,-172.675,85.953,-172.957
C07969=1012.027,178.208,-132.318,-172.734,85.945,-173.018
C07970=1012.027,178.444,-132.344,-172.793,85.936,-173.079
C07971=1012.025,178.680,-132.368,-172.862,85.927,-173.150
C07972=1012.026,178.915,-132.393,-172.921,85.919,-173.211
C07973=1012.025,179.152,-132.418,-172.979,85.910,-173.271
C07974=1012.025,179.387,-132.442,-173.048,85.900,-173.342
C07975=1012.024,179.623,-132.467,-173.106,85.891,-173.401
C07976=1012.023,179.858,-132.491,-173.163,85.883,-173.461
C07977=1012.023,180.094,-132.517,-173.231,85.874,-173.530
C07978=1012.023,180.330,-132.542,-173.288,85.865,-173.588
C07979=1012.022,180.566,-132.566,-173.344,85.856,-173.647
C07980=1012.021,180.802,-132.591,-173.400,85.848,-173.705
C07981=1012.022,181.037,-132.616,-173.456,85.839,-173.763
C07982=1012.021,181.274,-132.641,-173.523,85.830,-173.831
C07983=1012.021,181.509,-132.665,-173.579,85.820,-173.890
C07984=1012.020,181.746,-132.690,-173.644,85.811,-173.956
C07985=1012.019,181.981,-132.716,-173.700,85.802,-174.015
C07986=1012.019,182.216,-132.740,-173.754,85.793,-174.071
C07987=1012.018,182.453,-132.765,-173.809,85.784,-174.128
C07988=1012.018,182.689,-132.790,-173.873,85.775,-174.194
C07989=1012.018,182.925,-132.815,-173.927,85.767,-174.250
C07990=1012.017,183.160,-132.840,-173.981,85.758,-174.305
C07991=1012.017,183.396,-132.864,-174.035,85.749,-174.361
C07992=1012.016,183.632,-132.890,-174.099,85.739,-174.427
C07993=1012.017,183.868,-132.915,-174.152,85.730,-174.482
C07994=1012.015,184.104,-132.939,-174.215,85.720,-174.547
C07995=1012.015,184.340,-132.965,-174.267,85.712,-174.601
C07996=1012.015,184.575,-132.990,-174.330,85.703,-174.665
C07997=1012.014,184.812,-133.014,-174.382,85.694,-174.719
C07998=1012.013,185.047,-133.039,-174.434,85.684,-174.774
C07999=1012.013,185.283,-133.064,-174.485,85.676,-174.828
C08000=1012.013,185.519,-133.090,-174.537,85.667,-174.881
C08001=1012.013,185.755,-133.114,-174.598,85.658,-174.943
C08002=1012.012,185.991,-133.139,-174.649,85.648,-174.997
C08003=1012.011,186.226,-133.164,-174.710,85.638,-175.060
C08004=1012.012,186.462,-133.189,-174.760,85.629,-175.112
C08005=1012.011,186.699,-133.214,-174.820,85.619,-175.174
C08006=1012.010,186.934,-133.239,-174.870,85.611,-175.226
C08007=1012.011,187.170,-133.264,-174.920,85.602,-175.278
C08008=1012.010,187.406,-133.290,-174.969,85.593,-175.330
C08009=1012.009,187.643,-133.314,-175.019,85.584,-175.382
C08010=1012.009,187.878,-133.339,-175.078,85.574,-175.442
C08011=1012.009,188.114,-133.364,-175.127,85.565,-175.494
C08012=1012.008,188.350,-133.390,-175.185,85.555,-175.553
C08013=1012.008,188.586,-133.414,-175.233,85.546,-175.605
C08014=1012.008,188.822,-133.440,-175.291,85.536,-175.664
C08015=1012.007,189.058,-133.465,-175.339,85.526,-175.715
C08016=1012.007,189.293,-133.490,-175.396,85.517,-175.774
C08017=1012.007,189.529,-133.515,-175.444,85.508,-175.823
C08018=1012.006,189.766,-133.540,-175.491,85.499,-175.873
C08019=1012.006,190.002,-133.565,-175.539,85.490,-175.923
C08020=1012.005,190.237,-133.590,-175.595,85.481,-175.980
C08021=1012.005,190.473,-133.615,-175.642,85.471,-176.030
C08022=1012.005,190.709,-133.640,-175.688,85.461,-176.079
C08023=1012.005,190.944,-133.666,-175.744,85.452,-176.136
C08024=1012.004,191.181,-133.690,-175.799,85.442,-176.193
C08025=1012.004,191.417,-133.715,-175.845,85.432,-176.242
C08026=1012.004,191.653,-133.741,-175.891,85.424,-176.290
C08027=1012.003,191.889,-133.766,-175.936,85.414,-176.338
C08028=1012.003,192.124,-133.791,-175.990,85.405,-176.393
C08029=1012.003,192.360,-133.817,-176.035,85.395,-176.441
C08030=1012.002,192.596,-133.842,-176.080,85.386,-176.488
C08031=1012.002,192.833,-133.866,-176.134,85.376,-176.544
C08032=1012.002,193.069,-133.892,-176.178,85.367,-176.591
C08033=1012.001,193.304,-133.917,-176.232,85.356,-176.646
C08034=1012.001,193.540,-133.943,-176.276,85.347,-176.693
C08035=1012.001,193.776,-133.967,-176.328,85.337,-176.748
C08036=1012.001,194.012,-133.993,-176.372,85.328,-176.794
C08037=1012.000,194.248,-134.018,-176.416,85.319,-176.839
C08038=1012.001,194.484,-134.043,-176.468,85.309,-176.893
C08039=1012.000,194.720,-134.069,-176.511,85.299,-176.939
C08040=1012.000,194.956,-134.094,-176.554,85.290,-176.984
C08041=1011.999,195.192,-134.119,-176.605,85.280,-177.037
C08042=1011.999,195.428,-134.144,-176.648,85.271,-177.083
C08043=1011.999,195.664,-134.169,-176.698,85.261,-177.136
C08044=1011.998,195.900,-134.195,-176.749,85.250,-177.188
C08045=1011.999,196.136,-134.220,-176.791,85.241,-177.233
C08046=1011.998,196.372,-134.245,-176.833,85.231,-177.277
C08047=1011.998,196.608,-134.271,-176.883,85.222,-177.329
C08048=1011.998,196.844,-134.296,-176.924,85.212,-177.373
C08049=1011.998,197.080,-134.321,-176.965,85.202,-177.417
C08050=1011.997,197.316,-134.347,-177.015,85.192,-177.468
C08051=1011.997,197.552,-134.372,-177.056,85.183,-177.511
C08052=1011.997,197.787,-134.397,-177.104,85.172,-177.563
C08053=1011.997,198.023,-134.422,-177.145,85.163,-177.606
C08054=1011.997,198.260,-134.448,-177.193,85.153,-177.657
C08055=1011.996,198.507,-134.475,-177.233,85.142,-177.700
C08056=1011.996,198.898,-134.517,-177.314,85.126,-177.783
C08057=1011.996,199.289,-134.558,-177.385,85.109,-177.858
C08058=1011.996,199.531,-134.585,-177.424,85.100,-177.900
C08059=1011.996,199.760,-134.609,-177.471,85.090,-177.950
C08060=1011.995,199.992,-134.635,-177.510,85.080,-177.991
C08061=1011.995,200.234,-134.661,-177.557,85.070,-178.040
C08062=1011.995,200.487,-134.688,-177.595,85.059,-178.082
C08063=1011.995,200.743,-134.715,-177.642,85.049,-178.130
C08064=1011.995,200.981,-134.741,-177.688,85.039,-178.179
C08065=1011.995,201.205,-134.765,-177.726,85.029,-178.219
C08066=1011.994,201.422,-134.789,-177.764,85.020,-178.260
///RCONF 0,0,0,0,1,0,0,0,0,0,0,0,0,0,0,0,0,0,0,0,0,0,0,0
C08067=1011.994,201.838,-134.833,-177.840,85.002,-178.339
C08068=1011.994,202.044,-134.855,-177.869,84.994,-178.372
C08069=1011.994,202.262,-134.879,-177.906,84.984,-178.412
C08070=1011.999,203.513,-135.016,-174.538,84.971,-175.534
C08071=1012.001,203.759,-135.043,-174.573,84.962,-175.572
C08072=1012.003,204.003,-135.069,-174.624,84.952,-175.625
C08073=1012.005,204.246,-135.096,-174.667,84.943,-175.671
C08074=1012.007,204.491,-135.123,-174.709,84.933,-175.717
C08075=1012.009,204.735,-135.149,-174.752,84.923,-175.762
C08076=1012.011,204.980,-135.175,-174.794,84.914,-175.807
C08077=1012.013,205.223,-135.202,-174.836,84.904,-175.851
C08078=1012.015,205.467,-135.228,-174.878,84.895,-175.896
C08079=1012.017,205.711,-135.255,-174.919,84.884,-175.941
C08080=1012.019,205.955,-135.282,-174.961,84.875,-175.985
C08081=1012.021,206.199,-135.308,-175.002,84.865,-176.029
C08082=1012.023,206.442,-135.334,-175.035,84.857,-176.066
C08083=1012.025,206.685,-135.361,-175.076,84.847,-176.109
C08084=1012.027,206.928,-135.387,-175.117,84.838,-176.153
C08085=1012.029,207.171,-135.414,-175.158,84.828,-176.196
C08086=1012.031,207.414,-135.440,-175.198,84.818,-176.240
C08087=1012.034,207.657,-135.467,-175.238,84.808,-176.283
C08088=1012.036,207.899,-135.493,-175.279,84.799,-176.326
C08089=1012.038,208.142,-135.519,-175.319,84.789,-176.369
C08090=1012.040,208.385,-135.546,-175.358,84.780,-176.412
C08091=1012.042,208.627,-135.572,-175.398,84.770,-176.454
C08092=1012.044,208.870,-135.598,-175.438,84.761,-176.496
C08093=1012.047,209.112,-135.626,-175.477,84.751,-176.538
C08094=1012.048,209.355,-135.652,-175.516,84.742,-176.580
C08095=1012.051,209.597,-135.678,-175.555,84.732,-176.622
C08096=1012.053,209.839,-135.704,-175.586,84.723,-176.657
C08097=1012.055,210.082,-135.732,-175.625,84.714,-176.698
C08098=1012.057,210.324,-135.757,-175.664,84.704,-176.740
C08099=1012.060,210.567,-135.784,-175.702,84.695,-176.781
C08100=1012.062,210.810,-135.811,-175.740,84.685,-176.822
C08101=1012.064,211.052,-135.838,-175.779,84.676,-176.863
C08102=1012.066,211.295,-135.864,-175.817,84.666,-176.903
C08103=1012.068,211.538,-135.890,-175.854,84.657,-176.944
C08104=1012.071,211.780,-135.917,-175.884,84.648,-176.978
C08105=1012.073,212.023,-135.944,-175.922,84.638,-177.018
C08106=1012.075,212.266,-135.970,-175.959,84.629,-177.058
C08107=1012.078,212.510,-135.997,-175.997,84.619,-177.098
C08108=1012.080,212.753,-136.024,-176.034,84.610,-177.138
C08109=1012.082,212.996,-136.051,-176.063,84.601,-177.171
C08110=1012.084,213.241,-136.077,-176.100,84.590,-177.211
C08111=1012.086,213.485,-136.104,-176.137,84.581,-177.250
C08112=1012.089,213.728,-136.131,-176.173,84.571,-177.290
C08113=1012.091,213.973,-136.158,-176.210,84.562,-177.329
C08114=1012.093,214.217,-136.185,-176.239,84.553,-177.361
C08115=1012.095,214.461,-136.212,-176.275,84.543,-177.400
C08116=1012.098,214.706,-136.239,-176.311,84.534,-177.439
C08117=1012.100,214.951,-136.265,-176.347,84.524,-177.478
C08118=1012.103,215.196,-136.292,-176.382,84.514,-177.516
C08119=1012.105,215.441,-136.320,-176.410,84.505,-177.548
C08120=1012.107,215.687,-136.347,-176.446,84.496,-177.586
C08121=1012.109,215.932,-136.374,-176.481,84.486,-177.624
C08122=1012.112,216.178,-136.401,-176.509,84.477,-177.655
C08123=1012.114,216.423,-136.428,-176.544,84.468,-177.693
C08124=1012.117,216.670,-136.455,-176.579,84.458,-177.731
C08125=1012.119,216.918,-136.482,-176.614,84.449,-177.769
C08126=1012.121,217.173,-136.510,-176.649,84.438,-177.806
C08127=1012.124,217.432,-136.539,-176.690,84.428,-177.850
C08128=1012.127,217.697,-136.568,-176.725,84.418,-177.888
C08129=1012.129,217.977,-136.599,-176.759,84.408,-177.926
C08130=1012.132,218.268,-136.631,-176.800,84.396,-177.970
C08131=1012.135,218.560,-136.663,-176.833,84.385,-178.008
C08132=1012.138,218.857,-136.697,-176.866,84.374,-178.045
C08133=1012.141,219.160,-136.730,-176.907,84.362,-178.089
C08134=1012.144,219.457,-136.763,-176.940,84.351,-178.126
C08135=1012.147,219.737,-136.795,-176.973,84.340,-178.163
C08136=1012.150,220.010,-136.825,-177.013,84.330,-178.206
C08137=1012.152,220.270,-136.853,-177.046,84.319,-178.242
C08138=1012.154,220.520,-136.881,-177.079,84.310,-178.278
C08139=1012.157,220.765,-136.908,-177.112,84.301,-178.313
C08140=1012.160,221.011,-136.936,-177.138,84.292,-178.342
C08141=1012.163,221.256,-136.963,-177.170,84.282,-178.378
C08142=1012.165,221.502,-136.990,-177.203,84.273,-178.413
C08143=1012.168,221.748,-137.017,-177.228,84.264,-178.442
C08144=1012.170,221.994,-137.045,-177.254,84.255,-178.470
C08145=1012.173,222.240,-137.072,-177.286,84.246,-178.505
C08146=1012.175,222.486,-137.099,-177.311,84.237,-178.534
C08147=1012.178,222.731,-137.126,-177.343,84.227,-178.568
C08148=1012.181,222.977,-137.154,-177.368,84.218,-178.597
C08149=1012.183,223.223,-137.181,-177.400,84.209,-178.631
C08150=1012.186,223.469,-137.209,-177.424,84.200,-178.659
C08151=1012.188,223.714,-137.236,-177.456,84.190,-178.694
C08152=1012.191,223.961,-137.263,-177.487,84.180,-178.728
C08153=1012.193,224.206,-137.291,-177.519,84.171,-178.762
C08154=1012.196,224.452,-137.319,-177.550,84.161,-178.796
C08155=1012.198,224.697,-137.346,-177.574,84.152,-178.824
C08156=1012.201,224.943,-137.373,-177.599,84.144,-178.851
C08157=1012.203,225.189,-137.400,-177.623,84.135,-178.879
C08158=1012.206,225.435,-137.428,-177.653,84.125,-178.912
C08159=1012.209,225.680,-137.456,-177.678,84.117,-178.939
C08160=1012.211,225.926,-137.483,-177.708,84.107,-178.973
C08161=1012.214,226.172,-137.510,-177.739,84.098,-179.006
C08162=1012.217,226.417,-137.538,-177.762,84.088,-179.033
C08163=1012.220,226.664,-137.566,-177.792,84.078,-179.066
C08164=1012.222,226.909,-137.593,-177.822,84.069,-179.099
C08165=1012.225,227.155,-137.621,-177.845,84.060,-179.126
C08166=1012.227,227.400,-137.648,-177.876,84.051,-179.158
C08167=1012.230,227.646,-137.676,-177.899,84.042,-179.185
C08168=1012.232,227.891,-137.703,-177.922,84.033,-179.211
C08169=1012.235,228.138,-137.731,-177.945,84.024,-179.238
C08170=1012.238,228.383,-137.759,-177.975,84.015,-179.270
C08171=1012.241,228.629,-137.786,-177.998,84.006,-179.296
C08172=1012.244,228.874,-137.814,-178.027,83.996,-179.329
C08173=1012.246,229.120,-137.841,-178.056,83.986,-179.361
C08174=1012.249,229.366,-137.869,-178.085,83.977,-179.393
C08175=1012.252,229.612,-137.897,-178.108,83.968,-179.418
C08176=1012.254,229.857,-137.924,-178.137,83.958,-179.450
C08177=1012.257,230.103,-137.952,-178.159,83.950,-179.476
C08178=1012.260,230.349,-137.980,-178.182,83.941,-179.501
C08179=1012.262,230.594,-138.007,-178.204,83.932,-179.527
C08180=1012.265,230.840,-138.035,-178.226,83.923,-179.552
C08181=1012.268,231.086,-138.063,-178.255,83.914,-179.583
C08182=1012.271,231.331,-138.090,-178.277,83.905,-179.609
C08183=1012.274,231.577,-138.118,-178.305,83.896,-179.640
C08184=1012.276,231.822,-138.146,-178.333,83.885,-179.671
C08185=1012.279,232.068,-138.174,-178.355,83.876,-179.696
C08186=1012.282,232.314,-138.202,-178.383,83.867,-179.727
C08187=1012.285,232.560,-138.229,-178.405,83.858,-179.752
C08188=1012.287,232.805,-138.257,-178.426,83.850,-179.776
C08189=1012.291,233.050,-138.285,-178.448,83.841,-179.801
C08190=1012.294,233.296,-138.312,-178.470,83.833,-179.826
C08191=1012.297,233.541,-138.340,-178.491,83.824,-179.850
C08192=1012.300,233.787,-138.368,-178.518,83.814,-179.881
C08193=1012.303,234.033,-138.395,-178.539,83.805,-179.905
C08194=1012.305,234.278,-138.423,-178.566,83.795,-179.935
C08195=1012.308,234.523,-138.451,-178.587,83.786,-179.960
C08196=1012.311,234.770,-138.479,-178.614,83.776,-179.990
C08197=1012.314,235.015,-138.507,-178.635,83.767,179.986
C08198=1012.317,235.260,-138.535,-178.656,83.759,179.962
C08199=1012.320,235.506,-138.563,-178.677,83.751,179.938
C08200=1012.323,235.752,-138.590,-178.698,83.742,179.914
C08201=1012.326,235.997,-138.619,-178.719,83.733,179.890
C08202=1012.328,236.242,-138.646,-178.746,83.724,179.861
C08203=1012.331,236.488,-138.675,-178.766,83.715,179.837
C08204=1012.334,236.734,-138.703,-178.793,83.706,179.808
C08205=1012.337,236.980,-138.730,-178.813,83.697,179.784
C08206=1012.340,237.225,-138.758,-178.839,83.687,179.755
C08207=1012.343,237.470,-138.786,-178.859,83.678,179.732
C08208=1012.346,237.716,-138.814,-178.879,83.669,179.708
C08209=1012.349,237.961,-138.843,-178.899,83.660,179.685
C08210=1012.352,238.207,-138.871,-178.920,83.652,179.662
C08211=1012.355,238.452,-138.898,-178.940,83.644,179.639
C08212=1012.358,238.698,-138.927,-178.960,83.635,179.616
C08213=1012.361,238.944,-138.954,-178.980,83.626,179.593
C08214=1012.364,239.189,-138.982,-179.005,83.617,179.564
C08215=1012.367,239.435,-139.010,-179.025,83.608,179.541
C08216=1012.370,239.681,-139.039,-179.050,83.598,179.513
C08217=1012.372,239.925,-139.066,-179.069,83.589,179.490
C08218=1012.376,240.171,-139.094,-179.095,83.579,179.462
C08219=1012.379,240.416,-139.122,-179.108,83.571,179.445
C08220=1012.383,240.662,-139.150,-179.128,83.563,179.422
C08221=1012.386,240.908,-139.179,-179.148,83.555,179.400
C08222=1012.389,241.153,-139.207,-179.167,83.546,179.377
C08223=1012.392,241.399,-139.235,-179.186,83.537,179.355
C08224=1012.395,241.644,-139.264,-179.205,83.528,179.333
C08225=1012.398,241.889,-139.292,-179.224,83.519,179.310
C08226=1012.401,242.134,-139.320,-179.249,83.510,179.283
C08227=1012.404,242.380,-139.348,-179.268,83.501,179.261
C08228=1012.407,242.625,-139.376,-179.292,83.492,179.233
C08229=1012.410,242.871,-139.404,-179.311,83.482,179.211
C08230=1012.413,243.117,-139.432,-179.330,83.474,179.189
C08231=1012.416,243.362,-139.461,-179.343,83.466,179.173
C08232=1012.420,243.608,-139.489,-179.362,83.458,179.151
C08233=1012.423,243.853,-139.518,-179.380,83.449,179.129
C08234=1012.426,244.098,-139.546,-179.399,83.441,179.108
C08235=1012.429,244.344,-139.574,-179.417,83.432,179.086
C08236=1012.432,244.590,-139.602,-179.442,83.423,179.059
C08237=1012.436,244.835,-139.631,-179.460,83.413,179.037
C08238=1012.438,245.079,-139.659,-179.478,83.404,179.016
C08239=1012.441,245.325,-139.687,-179.502,83.395,178.989
C08240=1012.445,245.571,-139.715,-179.520,83.386,178.968
C08241=1012.448,245.816,-139.744,-179.533,83.379,178.952
C08242=1012.451,246.061,-139.772,-179.551,83.370,178.931
C08243=1012.454,246.307,-139.800,-179.569,83.361,178.909
C08244=1012.458,246.552,-139.829,-179.587,83.353,178.888
C08245=1012.461,246.797,-139.857,-179.605,83.344,178.867
C08246=1012.464,247.043,-139.886,-179.623,83.335,178.846
C08247=1012.467,247.288,-139.914,-179.641,83.327,178.825
C08248=1012.470,247.534,-139.943,-179.658,83.318,178.804
C08249=1012.473,247.779,-139.971,-179.681,83.308,178.778
C08250=1012.477,248.024,-140.000,-179.698,83.299,178.758
C08251=1012.481,248.270,-140.028,-179.716,83.291,178.737
C08252=1012.484,248.515,-140.057,-179.728,83.283,178.721
C08253=1012.487,248.761,-140.085,-179.746,83.275,178.701
C08254=1012.491,249.006,-140.114,-179.764,83.266,178.680
C08255=1012.494,249.252,-140.142,-179.776,83.259,178.665
C08256=1012.497,249.497,-140.170,-179.793,83.250,178.644
C08257=1012.500,249.742,-140.199,-179.810,83.241,178.624
C08258=1012.503,249.988,-140.228,-179.833,83.231,178.598
C08259=1012.507,250.232,-140.256,-179.850,83.222,178.578
C08260=1012.511,250.478,-140.284,-179.866,83.213,178.558
C08261=1012.514,250.723,-140.313,-179.889,83.204,178.532
C08262=1012.517,250.968,-140.342,-179.901,83.197,178.517
C08263=1012.521,251.214,-140.370,-179.913,83.189,178.502
C08264=1012.525,251.459,-140.399,-179.930,83.181,178.482
C08265=1012.528,251.705,-140.427,-179.947,83.172,178.462
C08266=1012.531,251.950,-140.456,-179.958,83.164,178.447
C08267=1012.535,252.195,-140.485,-179.975,83.155,178.427
C08268=1012.538,252.440,-140.513,-179.992,83.147,178.407
C08269=1012.541,252.685,-140.542,179.992,83.138,178.387
C08270=1012.544,252.930,-140.571,179.970,83.128,178.363
C08271=1012.548,253.177,-140.600,179.954,83.119,178.343
C08272=1012.552,253.422,-140.628,179.937,83.111,178.323
C08273=1012.555,253.667,-140.657,179.926,83.103,178.309
C08274=1012.558,253.912,-140.686,179.909,83.095,178.289
C08275=1012.562,254.157,-140.714,179.897,83.088,178.274
C08276=1012.566,254.403,-140.744,179.882,83.079,178.255
C08277=1012.569,254.648,-140.773,179.865,83.070,178.235
C08278=1012.572,254.893,-140.801,179.854,83.062,178.221
C08279=1012.576,255.138,-140.830,179.838,83.053,178.202
C08280=1012.579,255.383,-140.858,179.816,83.044,178.177
C08281=1012.583,255.629,-140.888,179.801,83.035,178.158
C08282=1012.586,255.874,-140.917,179.785,83.026,178.139
C08283=1012.590,256.119,-140.945,179.769,83.018,178.120
C08284=1012.592,256.365,-140.974,179.758,83.010,178.106
C08285=1012.596,256.611,-141.003,179.747,83.003,178.091
C08286=1012.600,256.855,-141.032,179.730,82.995,178.072
C08287=1012.603,257.100,-141.061,179.720,82.987,178.058
C08288=1012.606,257.345,-141.090,179.704,82.979,178.039
C08289=1012.611,257.591,-141.119,179.688,82.969,178.020
C08290=1012.614,257.836,-141.148,179.672,82.961,178.001
C08291=1012.617,258.081,-141.177,179.657,82.952,177.983
C08292=1012.621,258.327,-141.206,179.642,82.943,177.964
C08293=1012.625,258.572,-141.235,179.627,82.934,177.945
C08294=1012.639,259.817,-141.389,177.894,82.859,176.513
C08295=1012.642,260.228,-141.443,177.357,82.848,176.079
C08296=1012.644,260.639,-141.498,176.740,82.803,175.560
C08297=1012.644,261.050,-141.554,176.178,82.777,175.099
C08298=1012.644,261.462,-141.613,175.621,82.753,174.645
C08299=1012.643,261.873,-141.671,174.996,82.695,174.117
C08300=1012.641,262.284,-141.732,174.450,82.671,173.674
C08301=1012.637,262.695,-141.794,173.878,82.630,173.201
C08302=1012.633,263.105,-141.859,173.351,82.614,172.779
C08303=1012.628,263.516,-141.922,172.772,82.564,172.299
C08304=1012.622,263.927,-141.990,172.249,82.544,171.880
C08305=1012.615,264.337,-142.058,171.703,82.510,171.437
C08306=1012.607,264.748,-142.126,171.127,82.450,170.959
C08307=1012.598,265.158,-142.198,170.622,82.438,170.561
C08308=1012.588,265.569,-142.270,170.075,82.391,170.116
C08309=1012.577,265.978,-142.343,169.537,82.341,169.677
///RCONF 0,0,0,0,0,0,0,0,0,0,0,0,0,0,0,0,0,0,0,0,0,0,0,0
C08310=1012.566,266.388,-142.418,169.007,82.301,169.250
C08311=1012.553,266.798,-142.495,168.497,82.271,168.844
C08312=1012.538,267.208,-142.572,167.980,82.232,168.430
C08313=1012.523,267.618,-142.652,167.456,82.179,168.007
C08314=1012.508,268.027,-142.734,166.957,82.158,167.617
C08315=1012.490,268.436,-142.815,166.441,82.102,167.202
C08316=1012.473,268.845,-142.899,165.939,82.062,166.804
C08317=1012.454,269.254,-142.985,165.441,82.027,166.414
C08318=1012.433,269.663,-143.070,164.935,81.957,166.006
C08319=1012.412,270.072,-143.158,164.449,81.920,165.626
C08320=1012.390,270.480,-143.247,163.958,81.864,165.237
C08321=1012.367,270.888,-143.340,163.476,81.838,164.865
C08322=1012.342,271.296,-143.432,162.993,81.775,164.484
C08323=1012.318,271.704,-143.526,162.517,81.737,164.116
C08324=1012.291,272.112,-143.621,162.044,81.686,163.748
C08325=1012.263,272.519,-143.718,161.576,81.630,163.384
C08326=1012.236,272.927,-143.817,161.111,81.590,163.027
C08327=1012.206,273.334,-143.916,160.654,81.516,162.671
C08328=1012.176,273.741,-144.018,160.194,81.472,162.319
C08329=1012.144,274.147,-144.121,159.738,81.423,161.972
C08330=1012.112,274.554,-144.226,159.284,81.371,161.626
C08331=1012.078,274.960,-144.331,158.840,81.305,161.287
C08332=1012.043,275.367,-144.438,158.398,81.250,160.952
C08333=1012.008,275.773,-144.548,157.954,81.199,160.618
C08334=1011.971,276.178,-144.659,157.513,81.140,160.287
C08335=1011.933,276.584,-144.771,157.082,81.079,159.964
C08336=1011.894,276.988,-144.884,156.652,81.017,159.642
C08337=1011.854,277.394,-144.999,156.222,80.960,159.323
C08338=1011.812,277.798,-145.116,155.806,80.890,159.014
C08339=1011.791,278.001,-145.176,155.583,80.870,158.851
C08340=1011.770,278.202,-145.236,155.366,80.845,158.691
C08341=1011.749,278.405,-145.295,155.160,80.810,158.540
C08342=1011.726,278.607,-145.355,154.964,80.765,158.395
C08343=1011.704,278.809,-145.416,154.756,80.734,158.243
C08344=1011.682,279.011,-145.477,154.549,80.701,158.092
C08345=1011.659,279.212,-145.538,154.343,80.670,157.942
C08346=1011.636,279.414,-145.600,154.128,80.648,157.786
C08347=1011.613,279.615,-145.662,153.924,80.616,157.639
C08348=1011.589,279.817,-145.725,153.729,80.575,157.497
C08349=1011.566,280.019,-145.788,153.535,80.534,157.357
C08350=1011.542,280.220,-145.852,153.319,80.511,157.202
C08351=1011.517,280.421,-145.916,153.113,80.479,157.054
C08352=1011.492,280.623,-145.979,152.923,80.438,156.918
C08353=1011.467,280.825,-146.043,152.739,80.391,156.786
C08354=1011.441,281.025,-146.108,152.529,80.361,156.637
C08355=1011.416,281.226,-146.174,152.336,80.323,156.499
C08356=1011.390,281.427,-146.240,152.138,80.287,156.359
C08357=1011.364,281.627,-146.306,151.929,80.257,156.211
C08358=1011.338,281.829,-146.373,151.734,80.220,156.073
C08359=1011.311,282.029,-146.440,151.554,80.172,155.947
C08360=1011.284,282.230,-146.508,151.357,80.135,155.809
C08361=1011.257,282.430,-146.575,151.168,80.093,155.677
C08362=1011.229,282.631,-146.644,150.970,80.058,155.539
C08363=1011.201,282.831,-146.712,150.776,80.018,155.404
C08364=1011.173,283.031,-146.782,150.588,79.977,155.274
C08365=1011.145,283.231,-146.852,150.385,79.944,155.133
C08366=1011.115,283.431,-146.921,150.199,79.900,155.005
C08367=1011.086,283.631,-146.992,150.020,79.855,154.883
C08368=1011.057,283.830,-147.063,149.817,79.822,154.743
C08369=1011.027,284.031,-147.134,149.632,79.778,154.617
C08370=1010.997,284.230,-147.205,149.457,79.728,154.499
C08371=1010.966,284.429,-147.278,149.266,79.689,154.369
C08372=1010.935,284.629,-147.350,149.086,79.643,154.249
C08373=1010.904,284.828,-147.423,148.891,79.607,154.116
C08374=1010.873,285.027,-147.497,148.710,79.561,153.995
C08375=1010.842,285.226,-147.571,148.529,79.517,153.874
C08376=1010.810,285.425,-147.646,148.330,79.481,153.741
C08377=1010.777,285.623,-147.721,148.152,79.435,153.623
C08378=1010.744,285.823,-147.796,147.990,79.379,153.518
C08379=1010.711,286.021,-147.872,147.810,79.334,153.400
C08380=1010.678,286.219,-147.947,147.636,79.286,153.286
C08381=1010.645,286.417,-148.024,147.454,79.242,153.167
C08382=1010.610,286.615,-148.101,147.278,79.194,153.052
C08383=1010.576,286.813,-148.179,147.101,79.145,152.939
C08384=1010.542,287.012,-148.258,146.906,79.106,152.811
C08385=1010.506,287.208,-148.337,146.730,79.057,152.698
C08386=1010.472,287.407,-148.415,146.577,78.998,152.603
C08387=1010.436,287.604,-148.494,146.392,78.953,152.485
C08388=1010.400,287.801,-148.574,146.206,78.908,152.366
C08389=1010.364,287.998,-148.654,146.041,78.852,152.263
C08390=1010.327,288.196,-148.734,145.893,78.790,152.174
C08391=1010.290,288.392,-148.816,145.709,78.743,152.057
C08392=1010.253,288.589,-148.898,145.549,78.686,151.960
C08393=1010.215,288.786,-148.980,145.368,78.638,151.846
C08394=1010.177,288.982,-149.064,145.192,78.588,151.737
C08395=1010.139,289.179,-149.147,145.038,78.527,151.646
C08396=1010.100,289.375,-149.230,144.877,78.469,151.550
C08397=1010.061,289.571,-149.314,144.713,78.412,151.451
C08398=1010.022,289.766,-149.399,144.545,78.359,151.350
C08399=1009.982,289.962,-149.485,144.383,78.300,151.254
C08400=1009.942,290.157,-149.570,144.216,78.245,151.155
C08401=1009.902,290.353,-149.656,144.052,78.187,151.058
C08402=1009.860,290.548,-149.743,143.897,78.126,150.968
C08403=1009.819,290.743,-149.830,143.721,78.072,150.864
C08404=1009.778,290.938,-149.918,143.570,78.009,150.779
C08405=1009.735,291.132,-150.006,143.407,77.949,150.685
C08406=1009.693,291.327,-150.096,143.244,77.891,150.591
C08407=1009.650,291.521,-150.184,143.101,77.822,150.514
C08408=1009.608,291.715,-150.275,142.938,77.761,150.422
C08409=1009.564,291.909,-150.364,142.790,77.695,150.341
C08410=1009.521,292.103,-150.456,142.619,77.638,150.244
C08411=1009.476,292.296,-150.547,142.475,77.569,150.167
C08412=1009.431,292.489,-150.639,142.306,77.511,150.072
C08413=1009.386,292.682,-150.732,142.141,77.449,149.982
C08414=1009.341,292.875,-150.825,142.007,77.376,149.913
C08415=1009.295,293.068,-150.918,141.864,77.306,149.840
C08416=1009.249,293.260,-151.012,141.716,77.237,149.762
C08417=1009.202,293.452,-151.108,141.559,77.171,149.680
C08418=1009.155,293.644,-151.203,141.416,77.101,149.607
C08419=1009.108,293.835,-151.298,141.261,77.033,149.527
C08420=1009.060,294.027,-151.394,141.113,76.962,149.452
C08421=1009.012,294.219,-151.491,140.977,76.886,149.387
C08422=1008.963,294.410,-151.589,140.818,76.820,149.304
C08423=1008.914,294.601,-151.687,140.689,76.741,149.245
C08424=1008.864,294.791,-151.786,140.534,76.673,149.167
C08425=1008.814,294.982,-151.885,140.397,76.597,149.103
C08426=1008.765,295.172,-151.985,140.260,76.519,149.040
C08427=1008.714,295.362,-152.085,140.127,76.441,148.980
C08428=1008.663,295.551,-152.186,139.973,76.369,148.905
C08429=1008.611,295.741,-152.288,139.846,76.288,148.850
C08430=1008.559,295.930,-152.390,139.688,76.217,148.774
C08431=1008.506,296.118,-152.493,139.550,76.139,148.712
C08432=1008.454,296.307,-152.596,139.442,76.050,148.672
C08433=1008.400,296.495,-152.700,139.302,75.971,148.611
C08434=1008.347,296.683,-152.805,139.167,75.890,148.553
C08435=1008.293,296.871,-152.910,139.038,75.808,148.500
C08436=1008.237,297.058,-153.016,138.901,75.726,148.442
C08437=1008.182,297.245,-153.123,138.776,75.642,148.393
C08438=1008.127,297.432,-153.230,138.643,75.558,148.339
C08439=1008.071,297.618,-153.337,138.511,75.475,148.287
C08440=1008.014,297.804,-153.445,138.400,75.383,148.249
C08441=1007.958,297.991,-153.555,138.253,75.303,148.187
C08442=1007.900,298.177,-153.664,138.139,75.212,148.149
C08443=1007.842,298.361,-153.775,138.022,75.121,148.109
C08444=1007.784,298.547,-153.886,137.888,75.037,148.057
C08445=1007.725,298.732,-153.997,137.785,74.940,148.028
C08446=1007.666,298.916,-154.109,137.669,74.848,147.991
C08447=1007.606,299.100,-154.222,137.560,74.753,147.959
C08448=1007.545,299.284,-154.335,137.427,74.665,147.910
C08449=1007.485,299.467,-154.449,137.318,74.569,147.879
C08450=1007.423,299.650,-154.564,137.217,74.471,147.854
C08451=1007.363,299.833,-154.679,137.112,74.373,147.826
C08452=1007.300,300.015,-154.796,136.994,74.279,147.790
C08453=1007.237,300.197,-154.912,136.884,74.181,147.761
C08454=1007.174,300.379,-155.029,136.778,74.082,147.734
C08455=1007.110,300.560,-155.148,136.667,73.985,147.705
C08456=1007.046,300.741,-155.266,136.565,73.884,147.682
C08457=1006.982,300.922,-155.387,136.460,73.783,147.658
C08458=1006.917,301.101,-155.506,136.351,73.682,147.632
C08459=1006.852,301.281,-155.627,136.271,73.574,147.625
C08460=1006.785,301.460,-155.748,136.158,73.474,147.597
C08461=1006.718,301.639,-155.870,136.077,73.365,147.590
C08462=1006.652,301.817,-155.993,135.966,73.263,147.565
C08463=1006.584,301.996,-156.116,135.889,73.151,147.562
C08464=1006.516,302.173,-156.241,135.790,73.045,147.546
C08465=1006.447,302.351,-156.366,135.692,72.939,147.530
C08466=1006.377,302.528,-156.491,135.609,72.827,147.525
C08467=1006.308,302.705,-156.618,135.504,72.723,147.505
C08468=1006.237,302.880,-156.745,135.419,72.611,147.499
C08469=1006.167,303.056,-156.873,135.348,72.495,147.504
C08470=1006.096,303.231,-157.001,135.269,72.381,147.502
C08471=1006.024,303.405,-157.130,135.176,72.271,147.493
C08472=1005.952,303.580,-157.260,135.097,72.156,147.492
C08473=1005.879,303.753,-157.390,135.016,72.041,147.491
C08474=1005.806,303.926,-157.522,134.934,71.927,147.490
C08475=1005.732,304.099,-157.654,134.857,71.811,147.492
C08476=1005.658,304.272,-157.786,134.780,71.694,147.495
C08477=1005.583,304.444,-157.919,134.697,71.578,147.494
C08478=1005.508,304.615,-158.053,134.645,71.454,147.513
C08479=1005.431,304.785,-158.188,134.559,71.338,147.511
C08480=1005.355,304.956,-158.322,134.507,71.212,147.531
C08481=1005.278,305.125,-158.460,134.421,71.097,147.530
C08482=1005.200,305.295,-158.596,134.371,70.970,147.551
C08483=1005.122,305.464,-158.734,134.300,70.849,147.560
C08484=1005.043,305.632,-158.872,134.230,70.727,147.570
C08485=1004.964,305.800,-159.011,134.173,70.601,147.588
C08486=1004.885,305.966,-159.151,134.095,70.482,147.593
C08487=1004.804,306.133,-159.291,134.038,70.356,147.611
C08488=1004.723,306.300,-159.432,133.994,70.226,147.638
C08489=1004.643,306.465,-159.573,133.942,70.098,147.660
C08490=1004.560,306.629,-159.716,133.877,69.974,147.674
C08491=1004.478,306.794,-159.859,133.824,69.846,147.696
C08492=1004.395,306.957,-160.003,133.769,69.719,147.716
C08493=1004.312,307.121,-160.147,133.713,69.591,147.737
C08494=1004.228,307.282,-160.293,133.662,69.462,147.761
C08495=1004.144,307.445,-160.438,133.613,69.332,147.786
C08496=1004.058,307.606,-160.586,133.556,69.204,147.806
C08497=1003.973,307.766,-160.732,133.532,69.068,147.845
C08498=1003.887,307.927,-160.880,133.464,68.942,147.860
C08499=1003.800,308.086,-161.029,133.433,68.806,147.895
C08500=1003.713,308.245,-161.178,133.382,68.676,147.920
C08501=1003.626,308.403,-161.328,133.340,68.543,147.950
C08502=1003.537,308.560,-161.479,133.312,68.406,147.988
C08503=1003.448,308.718,-161.630,133.274,68.273,148.020
C08504=1003.359,308.874,-161.783,133.225,68.142,148.046
C08505=1003.270,309.029,-161.936,133.195,68.005,148.083
C08506=1003.179,309.184,-162.089,133.146,67.875,148.109
C08507=1003.088,309.338,-162.244,133.103,67.742,148.138
C08508=1002.997,309.492,-162.397,133.097,67.601,148.187
C08509=1002.889,309.670,-162.579,133.056,67.444,148.227
C08510=1002.781,309.848,-162.762,133.017,67.287,148.267
C08511=1002.672,310.025,-162.946,132.994,67.125,148.317
C08512=1002.563,310.200,-163.130,132.945,66.970,148.352
C08513=1002.668,309.793,-163.338,117.545,69.709,139.642
C08514=1002.761,309.643,-163.181,117.476,69.886,139.483
C08515=1002.853,309.494,-163.027,117.410,70.062,139.326
C08516=1002.944,309.342,-162.871,117.337,70.239,139.163
C08517=1003.036,309.190,-162.717,117.271,70.413,139.005
C08518=1003.126,309.038,-162.564,117.168,70.593,138.822
C08519=1003.216,308.885,-162.411,117.106,70.768,138.664
C08520=1003.305,308.732,-162.259,117.055,70.940,138.513
C08521=1003.395,308.577,-162.107,116.973,71.116,138.341
C08522=1003.483,308.423,-161.956,116.918,71.289,138.185
C08523=1003.571,308.266,-161.806,116.844,71.463,138.016
C08524=1003.659,308.110,-161.657,116.756,71.639,137.838
C08525=1003.745,307.953,-161.508,116.684,71.812,137.669
C08526=1003.832,307.796,-161.360,116.621,71.985,137.506
C08527=1003.919,307.636,-161.212,116.532,72.159,137.325
C08528=1004.004,307.478,-161.064,116.489,72.327,137.174
C08529=1004.089,307.318,-160.918,116.388,72.501,136.983
C08530=1004.173,307.158,-160.773,116.326,72.671,136.818
C08531=1004.257,306.998,-160.628,116.253,72.841,136.646
C08532=1004.340,306.836,-160.484,116.181,73.009,136.473
C08533=1004.423,306.675,-160.340,116.114,73.176,136.304
C08534=1004.505,306.512,-160.197,116.045,73.343,136.133
C08535=1004.587,306.349,-160.055,115.970,73.510,135.957
C08536=1004.668,306.185,-159.913,115.908,73.675,135.791
C08537=1004.749,306.021,-159.773,115.830,73.841,135.611
C08538=1004.829,305.856,-159.633,115.735,74.009,135.420
C08539=1004.908,305.690,-159.494,115.659,74.173,135.241
C08540=1004.988,305.525,-159.355,115.609,74.333,135.081
C08541=1005.066,305.358,-159.218,115.528,74.496,134.899
C08542=1005.145,305.191,-159.079,115.462,74.657,134.727
C08543=1005.222,305.024,-158.943,115.398,74.817,134.555
C08544=1005.299,304.855,-158.808,115.299,74.981,134.358
C08545=1005.375,304.687,-158.672,115.251,75.136,134.198
C08546=1005.451,304.518,-158.538,115.152,75.298,134.001
C08547=1005.527,304.349,-158.404,115.100,75.452,133.838
C08548=1005.602,304.179,-158.271,114.999,75.613,133.637
C08549=1005.676,304.008,-158.138,114.936,75.766,133.466
C08550=1005.750,303.836,-158.007,114.864,75.920,133.288
C08551=1005.823,303.665,-157.876,114.790,76.074,133.108
C08552=1005.896,303.493,-157.746,114.725,76.225,132.933
C08553=1005.968,303.321,-157.616,114.656,76.376,132.757
C08554=1006.040,303.147,-157.487,114.579,76.527,132.575
C08555=1006.111,302.974,-157.359,114.522,76.675,132.407
C08556=1006.182,302.800,-157.232,114.440,76.824,132.220
C08557=1006.252,302.626,-157.105,114.343,76.975,132.021
C08558=1006.322,302.451,-156.979,114.268,77.122,131.838
C08559=1006.391,302.276,-156.853,114.225,77.264,131.682
C08560=1006.459,302.101,-156.728,114.140,77.411,131.491
C08561=1006.528,301.924,-156.604,114.078,77.553,131.321
C08562=1006.595,301.748,-156.481,114.017,77.694,131.150
C08563=1006.663,301.570,-156.359,113.911,77.840,130.942
C08564=1006.730,301.393,-156.236,113.868,77.977,130.786
C08565=1006.795,301.215,-156.115,113.769,78.119,130.585
C08566=1006.861,301.038,-155.994,113.721,78.255,130.425
C08567=1006.926,300.859,-155.875,113.614,78.397,130.217
C08568=1006.990,300.680,-155.755,113.554,78.532,130.048
C08569=1007.055,300.501,-155.636,113.490,78.665,129.876
C08570=1007.119,300.321,-155.519,113.413,78.800,129.693
C08571=1007.181,300.141,-155.401,113.352,78.932,129.523
C08572=1007.244,299.961,-155.284,113.281,79.064,129.346
C08573=1007.307,299.780,-155.168,113.210,79.195,129.168
C08574=1007.368,299.598,-155.052,113.158,79.323,129.006
C08575=1007.429,299.417,-154.939,113.078,79.453,128.821
C08576=1007.490,299.236,-154.824,112.983,79.584,128.623
C08577=1007.550,299.053,-154.711,112.905,79.711,128.441
C08578=1007.610,298.870,-154.598,112.872,79.833,128.296
C08579=1007.670,298.688,-154.486,112.783,79.960,128.104
C08580=1007.729,298.505,-154.374,112.712,80.084,127.928
C08581=1007.787,298.320,-154.264,112.604,80.210,127.720
C08582=1007.845,298.137,-154.154,112.566,80.328,127.573
C08583=1007.902,297.953,-154.044,112.486,80.451,127.389
C08584=1007.959,297.768,-153.935,112.398,80.572,127.199
C08585=1008.016,297.583,-153.827,112.380,80.685,127.070
C08586=1008.072,297.399,-153.719,112.279,80.806,126.869
C08587=1008.127,297.213,-153.612,112.222,80.921,126.707
C08588=1008.183,297.028,-153.505,112.160,81.036,126.540
C08589=1008.237,296.841,-153.400,112.089,81.151,126.366
C08590=1008.292,296.655,-153.295,112.031,81.263,126.205
C08591=1008.345,296.469,-153.190,111.963,81.376,126.034
C08592=1008.399,296.282,-153.086,111.895,81.487,125.864
C08593=1008.452,296.094,-152.982,111.846,81.596,125.710
C08594=1008.505,295.907,-152.880,111.713,81.712,125.482
C08595=1008.556,295.719,-152.778,111.648,81.821,125.315
C08596=1008.608,295.532,-152.676,111.634,81.923,125.195
C08597=1008.659,295.343,-152.575,111.536,82.033,125.000
C08598=1008.710,295.155,-152.474,111.506,82.135,124.865
C08599=1008.761,294.966,-152.375,111.418,82.242,124.680
C08600=1008.810,294.777,-152.276,111.336,82.347,124.499
C08601=1008.860,294.588,-152.177,111.252,82.452,124.317
C08602=1008.909,294.398,-152.079,111.225,82.550,124.188
C08603=1008.958,294.208,-151.982,111.110,82.656,123.978
C08604=1009.006,294.018,-151.884,111.075,82.754,123.842
C08605=1009.054,293.828,-151.788,110.973,82.856,123.646
C08606=1009.101,293.638,-151.692,110.913,82.954,123.487
C08607=1009.148,293.447,-151.597,110.862,83.050,123.339
C08608=1009.195,293.256,-151.502,110.781,83.148,123.162
C08609=1009.242,293.065,-151.408,110.730,83.243,123.013
C08610=1009.288,292.874,-151.314,110.654,83.338,122.842
C08611=1009.334,292.682,-151.221,110.548,83.435,122.644
C08612=1009.378,292.490,-151.129,110.424,83.534,122.428
C08613=1009.423,292.299,-151.036,110.389,83.623,122.297
C08614=1009.468,292.106,-150.945,110.366,83.712,122.176
C08615=1009.511,291.914,-150.854,110.259,83.805,121.978
C08616=1009.555,291.721,-150.764,110.246,83.891,121.868
C08617=1009.598,291.528,-150.674,110.144,83.983,121.675
C08618=1009.641,291.335,-150.584,110.089,84.071,121.526
C08619=1009.683,291.142,-150.496,109.950,84.164,121.299
C08620=1009.725,290.948,-150.407,109.904,84.249,121.161
C08621=1009.767,290.755,-150.319,109.833,84.335,120.998
C08622=1009.809,290.561,-150.232,109.716,84.425,120.792
C08623=1009.849,290.368,-150.145,109.704,84.505,120.686
C08624=1009.890,290.173,-150.058,109.596,84.592,120.490
C08625=1009.931,289.979,-149.973,109.523,84.676,120.326
C08626=1009.971,289.784,-149.887,109.462,84.758,120.176
C08627=1010.010,289.590,-149.803,109.373,84.841,119.999
C08628=1010.050,289.395,-149.718,109.320,84.921,119.856
C08629=1010.088,289.199,-149.634,109.221,85.003,119.671
C08630=1010.126,289.005,-149.551,109.112,85.085,119.475
C08631=1010.165,288.809,-149.470,108.961,85.169,119.240
C08632=1010.202,288.613,-149.387,108.915,85.246,119.105
C08633=1010.240,288.418,-149.304,108.902,85.321,119.002
C08634=1010.277,288.222,-149.223,108.771,85.401,118.787
C08635=1010.313,288.027,-149.142,108.751,85.474,118.679
C08636=1010.351,287.830,-149.062,108.545,85.559,118.391
C08637=1010.386,287.633,-148.982,108.405,85.637,118.168
C08638=1010.422,287.437,-148.902,108.383,85.710,118.058
C08639=1010.457,287.241,-148.823,108.357,85.781,117.944
C08640=1010.493,287.044,-148.745,108.152,85.862,117.660
C08641=1010.527,286.847,-148.666,108.056,85.935,117.481
C08642=1010.561,286.650,-148.588,108.089,86.002,117.425
C08643=1010.595,286.454,-148.511,107.979,86.076,117.232
C08644=1010.629,286.257,-148.434,107.890,86.148,117.060
C08645=1010.663,286.058,-148.358,107.832,86.217,116.918
C08646=1010.696,285.861,-148.282,107.711,86.289,116.716
C08647=1010.729,285.664,-148.207,107.625,86.359,116.548
C08648=1010.761,285.465,-148.132,107.386,86.434,116.232
C08649=1010.793,285.267,-148.058,107.267,86.504,116.033
C08650=1010.825,285.070,-147.983,107.295,86.567,115.975
C08651=1010.856,284.872,-147.910,107.200,86.636,115.799
C08652=1010.887,284.674,-147.837,107.053,86.705,115.573
C08653=1010.919,284.476,-147.764,107.065,86.768,115.502
C08654=1010.949,284.277,-147.691,106.909,86.837,115.267
C08655=1010.979,284.079,-147.619,106.847,86.902,115.124
C08656=1011.010,283.879,-147.548,106.611,86.973,114.810
C08657=1011.039,283.680,-147.477,106.463,87.039,114.584
C08658=1011.068,283.482,-147.407,106.460,87.101,114.498
C08659=1011.097,283.282,-147.337,106.265,87.169,114.226
C08660=1011.126,283.083,-147.267,106.085,87.235,113.968
C08661=1011.154,282.885,-147.197,106.076,87.295,113.878
C08662=1011.183,282.685,-147.128,105.923,87.360,113.646
C08663=1011.210,282.485,-147.060,105.797,87.423,113.442
C08664=1011.238,282.287,-146.991,105.722,87.484,113.289
C08665=1011.265,282.086,-146.924,105.526,87.548,113.016
C08666=1011.292,281.888,-146.857,105.397,87.610,112.808
C08667=1011.318,281.688,-146.790,105.026,87.678,112.364
C08668=1011.345,281.487,-146.725,104.852,87.739,112.113
C08669=1011.371,281.288,-146.658,104.862,87.795,112.044
C08670=1011.397,281.087,-146.592,104.724,87.855,111.828
C08671=1011.422,280.887,-146.527,104.475,87.918,111.504
C08672=1011.448,280.687,-146.462,104.449,87.973,111.401
C08673=1011.472,280.487,-146.399,103.971,88.040,110.850
C08674=1011.497,280.286,-146.334,103.610,88.102,110.415
C08675=1011.521,280.086,-146.271,103.453,88.159,110.183
C08676=1011.569,279.685,-146.145,103.142,88.273,109.719
C08677=1011.616,279.282,-146.021,102.448,88.390,108.880
C08678=1011.661,278.881,-145.897,102.274,88.498,108.552
C08679=1011.706,278.479,-145.776,101.639,88.610,107.770
C08680=1011.748,278.076,-145.658,100.303,88.730,106.291
C08681=1011.791,277.673,-145.539,100.220,88.830,106.055
C08682=1011.832,277.270,-145.422,98.846,88.944,104.536
C08683=1011.872,276.867,-145.308,97.789,89.051,103.332
C08684=1011.911,276.464,-145.195,96.145,89.159,101.542
C08685=1011.949,276.060,-145.083,94.016,89.265,99.269
C08686=1011.986,275.656,-144.973,91.318,89.369,96.426
C08687=1012.022,275.251,-144.864,88.341,89.468,93.304
C08688=1012.056,274.847,-144.756,83.465,89.566,88.283
C08689=1012.089,274.441,-144.652,74.008,89.659,78.685
C08690=1012.121,274.037,-144.547,61.182,89.737,65.716
C08691=1012.153,273.632,-144.444,40.422,89.795,44.811
C08692=1012.184,273.226,-144.343,11.933,89.815,16.178
C08693=1012.212,272.820,-144.245,-15.835,89.754,-11.726
C08694=1012.241,272.415,-144.145,-31.593,89.695,-27.627
C08695=1012.268,272.009,-144.050,-40.856,89.606,-37.029
///RCONF 0,0,0,0,1,0,0,0,0,0,0,0,0,0,0,0,0,0,0,0,0,0,0,0
C08696=1012.294,271.603,-143.955,-46.802,89.514,-43.116
C08697=1012.319,271.196,-143.861,-51.479,89.431,-47.936
C08698=1012.343,270.790,-143.769,-53.694,89.322,-50.288
C08699=1012.367,270.383,-143.678,-56.844,89.245,-53.582
C08700=1012.388,269.977,-143.589,-58.098,89.140,-54.974
C08701=1012.409,269.569,-143.500,-59.761,89.050,-56.778
C08702=1012.429,269.162,-143.415,-59.964,88.933,-57.116
C08703=1012.448,268.755,-143.330,-61.226,88.845,-58.519
C08704=1012.466,268.347,-143.246,-62.096,88.751,-59.528
C08705=1012.477,268.083,-143.193,-62.170,88.679,-59.690
C08706=1012.488,267.818,-143.141,-62.630,88.618,-60.241
C08707=1012.498,267.553,-143.087,-63.448,88.568,-61.152
C08708=1012.508,267.289,-143.037,-63.770,88.506,-61.564
C08709=1012.519,267.002,-142.982,-63.773,88.430,-61.660
C08710=1012.528,266.716,-142.927,-64.230,88.367,-62.216
C08711=1012.541,266.307,-142.851,-64.823,88.279,-62.947
C08712=1012.553,265.899,-142.776,-65.151,88.184,-63.413
C08713=1012.564,265.490,-142.703,-65.186,88.080,-63.583
C08714=1012.574,265.082,-142.632,-65.310,87.980,-63.844
C08715=1012.583,264.673,-142.559,-66.071,87.905,-64.745
C08716=1012.591,264.264,-142.492,-65.836,87.794,-64.644
C08717=1012.598,263.855,-142.424,-66.080,87.702,-65.024
C08718=1012.604,263.446,-142.358,-66.561,87.621,-65.644
C08719=1012.609,263.037,-142.293,-66.461,87.516,-65.678
C08720=1012.614,262.627,-142.229,-66.933,87.437,-66.290
C08721=1012.616,262.218,-142.167,-66.927,87.338,-66.418
C08722=1012.619,261.809,-142.107,-67.215,87.253,-66.843
C08723=1012.620,261.399,-142.049,-66.944,87.142,-66.705
C08724=1012.620,260.989,-141.991,-67.168,87.055,-67.064
C08725=1012.620,260.579,-141.934,-67.347,86.968,-67.379
C08726=1012.618,260.169,-141.881,-67.245,86.865,-67.411
C08727=1012.615,259.759,-141.825,-67.580,86.788,-67.883
C08728=1012.602,258.519,-141.672,-67.927,86.525,-68.632
C08729=1012.598,258.274,-141.643,-67.798,86.518,-68.501
C08730=1012.595,258.029,-141.614,-67.674,86.512,-68.374
C08731=1012.592,257.784,-141.585,-67.562,86.506,-68.260
C08732=1012.588,257.538,-141.557,-67.439,86.500,-68.134
C08733=1012.584,257.293,-141.528,-67.333,86.495,-68.025
C08734=1012.581,257.048,-141.499,-67.222,86.489,-67.912
C08735=1012.578,256.803,-141.470,-67.111,86.483,-67.800
C08736=1012.574,256.557,-141.441,-67.018,86.478,-67.704
C08737=1012.570,256.313,-141.412,-66.913,86.473,-67.596
C08738=1012.567,256.068,-141.383,-66.819,86.468,-67.501
C08739=1012.563,255.823,-141.354,-66.710,86.462,-67.389
C08740=1012.560,255.578,-141.325,-66.590,86.456,-67.267
C08741=1012.557,255.332,-141.297,-66.471,86.449,-67.145
C08742=1012.553,255.086,-141.268,-66.363,86.443,-67.035
C08743=1012.549,254.841,-141.239,-66.244,86.437,-66.913
C08744=1012.546,254.596,-141.210,-66.137,86.431,-66.804
C08745=1012.544,254.350,-141.181,-66.030,86.425,-66.695
C08746=1012.540,254.105,-141.152,-65.928,86.420,-66.590
C08747=1012.537,253.861,-141.123,-65.822,86.414,-66.482
C08748=1012.533,253.616,-141.094,-65.732,86.409,-66.390
C08749=1012.530,253.369,-141.066,-65.631,86.403,-66.286
C08750=1012.526,253.124,-141.037,-65.526,86.397,-66.179
C08751=1012.523,252.879,-141.008,-65.410,86.391,-66.060
C08752=1012.520,252.634,-140.980,-65.295,86.384,-65.942
C08753=1012.516,252.389,-140.951,-65.186,86.377,-65.833
C08754=1012.513,252.144,-140.922,-65.076,86.371,-65.719
C08755=1012.510,251.898,-140.894,-64.973,86.365,-65.614
C08756=1012.506,251.653,-140.865,-64.870,86.359,-65.509
C08757=1012.503,251.408,-140.837,-64.768,86.353,-65.404
C08758=1012.500,251.163,-140.808,-64.670,86.347,-65.304
C08759=1012.496,250.918,-140.779,-64.572,86.342,-65.203
C08760=1012.493,250.671,-140.751,-64.481,86.336,-65.111
C08761=1012.489,250.426,-140.722,-64.369,86.329,-64.996
C08762=1012.486,250.181,-140.694,-64.258,86.323,-64.882
C08763=1012.483,249.936,-140.665,-64.157,86.316,-64.780
C08764=1012.480,249.690,-140.637,-64.047,86.310,-64.666
C08765=1012.476,249.445,-140.608,-63.937,86.303,-64.554
C08766=1012.473,249.200,-140.580,-63.837,86.297,-64.452
C08767=1012.470,248.955,-140.551,-63.738,86.290,-64.351
C08768=1012.466,248.709,-140.523,-63.639,86.284,-64.250
C08769=1012.463,248.463,-140.494,-63.545,86.279,-64.153
C08770=1012.460,248.218,-140.465,-63.457,86.272,-64.064
C08771=1012.457,247.973,-140.437,-63.363,86.267,-63.967
C08772=1012.453,247.728,-140.408,-63.256,86.260,-63.857
C08773=1012.450,247.482,-140.380,-63.144,86.252,-63.744
C08774=1012.447,247.237,-140.352,-63.038,86.246,-63.634
C08775=1012.444,246.992,-140.323,-62.941,86.239,-63.536
C08776=1012.441,246.747,-140.295,-62.835,86.232,-63.427
C08777=1012.439,246.501,-140.267,-62.740,86.226,-63.329
C08778=1012.435,246.256,-140.238,-62.644,86.219,-63.232
C08779=1012.432,246.010,-140.210,-62.553,86.214,-63.138
C08780=1012.429,245.765,-140.181,-62.458,86.207,-63.041
C08781=1012.426,245.520,-140.153,-62.367,86.202,-62.948
C08782=1012.423,245.274,-140.124,-62.273,86.195,-62.852
C08783=1012.420,245.029,-140.096,-62.170,86.188,-62.745
C08784=1012.416,244.783,-140.068,-62.063,86.180,-62.637
C08785=1012.413,244.538,-140.039,-61.960,86.173,-62.531
C08786=1012.410,244.292,-140.011,-61.858,86.166,-62.426
C08787=1012.407,244.047,-139.983,-61.765,86.160,-62.332
C08788=1012.404,243.802,-139.955,-61.673,86.153,-62.238
C08789=1012.401,243.556,-139.927,-61.582,86.147,-62.144
C08790=1012.398,243.311,-139.899,-61.484,86.140,-62.043
C08791=1012.395,243.066,-139.870,-61.403,86.134,-61.960
C08792=1012.392,242.820,-139.842,-61.312,86.128,-61.868
C08793=1012.388,242.575,-139.813,-61.212,86.120,-61.765
C08794=1012.385,242.329,-139.785,-61.112,86.113,-61.662
C08795=1012.382,242.083,-139.757,-61.013,86.106,-61.560
C08796=1012.380,241.838,-139.729,-60.911,86.098,-61.456
C08797=1012.377,241.593,-139.701,-60.822,86.092,-61.365
C08798=1012.373,241.347,-139.673,-60.724,86.085,-61.265
C08799=1012.370,241.102,-139.645,-60.635,86.078,-61.174
C08800=1012.367,240.856,-139.617,-60.547,86.071,-61.084
C08801=1012.365,240.611,-139.589,-60.462,86.065,-60.996
C08802=1012.362,240.366,-139.561,-60.375,86.058,-60.907
C08803=1012.358,240.120,-139.532,-60.288,86.052,-60.818
C08804=1012.355,239.874,-139.504,-60.191,86.044,-60.719
C08805=1012.352,239.629,-139.476,-60.096,86.037,-60.620
C08806=1012.350,239.384,-139.448,-59.997,86.029,-60.520
C08807=1012.347,239.138,-139.420,-59.902,86.022,-60.422
C08808=1012.343,238.893,-139.392,-59.807,86.015,-60.325
C08809=1012.340,238.647,-139.364,-59.722,86.008,-60.237
C08810=1012.338,238.402,-139.336,-59.628,86.001,-60.141
C08811=1012.335,238.157,-139.308,-59.543,85.994,-60.054
C08812=1012.332,237.911,-139.280,-59.459,85.987,-59.968
C08813=1012.329,237.665,-139.252,-59.375,85.980,-59.882
C08814=1012.326,237.420,-139.224,-59.294,85.974,-59.798
C08815=1012.323,237.174,-139.196,-59.198,85.966,-59.701
C08816=1012.320,236.929,-139.168,-59.106,85.959,-59.606
C08817=1012.317,236.683,-139.140,-59.012,85.950,-59.510
C08818=1012.314,236.438,-139.112,-58.920,85.943,-59.415
C08819=1012.312,236.192,-139.085,-58.829,85.936,-59.322
C08820=1012.309,235.946,-139.057,-58.747,85.929,-59.238
C08821=1012.306,235.702,-139.029,-58.657,85.921,-59.145
C08822=1012.303,235.456,-139.001,-58.575,85.914,-59.061
C08823=1012.300,235.210,-138.972,-58.494,85.907,-58.978
C08824=1012.297,234.964,-138.945,-58.414,85.900,-58.896
C08825=1012.294,234.719,-138.917,-58.324,85.893,-58.804
C08826=1012.291,234.474,-138.889,-58.235,85.886,-58.712
C08827=1012.289,234.227,-138.861,-58.144,85.877,-58.619
C08828=1012.286,233.982,-138.834,-58.056,85.870,-58.528
C08829=1012.283,233.737,-138.806,-57.966,85.861,-58.436
C08830=1012.281,233.491,-138.778,-57.887,85.854,-58.355
C08831=1012.278,233.246,-138.750,-57.800,85.847,-58.265
C08832=1012.274,233.000,-138.722,-57.713,85.839,-58.176
C08833=1012.272,232.755,-138.695,-57.634,85.832,-58.096
C08834=1012.269,232.509,-138.667,-57.557,85.825,-58.016
C08835=1012.266,232.263,-138.639,-57.479,85.818,-57.936
C08836=1012.264,232.018,-138.612,-57.393,85.811,-57.848
C08837=1012.261,231.772,-138.583,-57.308,85.803,-57.760
C08838=1012.258,231.526,-138.556,-57.220,85.795,-57.671
C08839=1012.255,231.281,-138.528,-57.136,85.787,-57.583
C08840=1012.253,231.035,-138.501,-57.049,85.779,-57.495
C08841=1012.250,230.790,-138.473,-56.965,85.771,-57.408
C08842=1012.247,230.544,-138.445,-56.881,85.763,-57.321
C08843=1012.245,230.299,-138.418,-56.806,85.756,-57.244
C08844=1012.242,230.053,-138.390,-56.731,85.749,-57.167
C08845=1012.239,229.807,-138.362,-56.648,85.742,-57.081
C08846=1012.237,229.562,-138.335,-56.573,85.734,-57.005
C08847=1012.234,229.316,-138.307,-56.489,85.726,-56.919
C08848=1012.231,229.071,-138.280,-56.407,85.718,-56.834
C08849=1012.229,228.824,-138.252,-56.323,85.710,-56.748
C08850=1012.227,228.579,-138.224,-56.241,85.702,-56.664
C08851=1012.224,228.333,-138.196,-56.158,85.693,-56.579
C08852=1012.221,228.087,-138.168,-56.077,85.686,-56.496
C08853=1012.219,227.842,-138.141,-55.997,85.678,-56.413
C08854=1012.216,227.596,-138.114,-55.925,85.671,-56.338
C08855=1012.213,227.351,-138.086,-55.853,85.663,-56.264
C08856=1012.210,227.104,-138.058,-55.773,85.656,-56.182
C08857=1012.208,226.859,-138.031,-55.701,85.648,-56.109
C08858=1012.205,226.613,-138.003,-55.612,85.639,-56.017
C08859=1012.203,226.368,-137.976,-55.532,85.631,-55.935
C08860=1012.200,226.122,-137.949,-55.453,85.623,-55.853
C08861=1012.198,225.877,-137.921,-55.373,85.614,-55.772
C08862=1012.195,225.630,-137.893,-55.295,85.607,-55.691
C08863=1012.193,225.385,-137.866,-55.217,85.599,-55.611
C08864=1012.190,225.139,-137.839,-55.146,85.590,-55.538
C08865=1012.187,224.894,-137.811,-55.069,85.583,-55.458
C08866=1012.184,224.648,-137.784,-55.000,85.575,-55.387
C08867=1012.182,224.402,-137.757,-54.923,85.568,-55.308
C08868=1012.180,224.157,-137.729,-54.855,85.560,-55.238
C08869=1012.177,223.910,-137.702,-54.769,85.551,-55.150
C08870=1012.175,223.665,-137.674,-54.692,85.542,-55.071
C08871=1012.172,223.419,-137.647,-54.616,85.534,-54.992
C08872=1012.170,223.174,-137.620,-54.540,85.526,-54.914
C08873=1012.167,222.928,-137.592,-54.465,85.518,-54.836
C08874=1012.165,222.682,-137.565,-54.388,85.509,-54.758
C08875=1012.162,222.436,-137.538,-54.314,85.501,-54.681
C08876=1012.160,222.190,-137.511,-54.247,85.494,-54.613
C08877=1012.157,221.944,-137.483,-54.174,85.486,-54.536
C08878=1012.154,221.699,-137.455,-54.107,85.478,-54.468
C08879=1012.152,221.454,-137.428,-54.033,85.469,-54.392
C08880=1012.149,221.207,-137.401,-53.960,85.461,-54.316
C08881=1012.147,220.962,-137.374,-53.885,85.453,-54.240
C08882=1012.145,220.716,-137.347,-53.813,85.445,-54.165
C08883=1012.142,220.470,-137.319,-53.748,85.437,-54.098
C08884=1012.140,220.221,-137.291,-53.675,85.428,-54.023
C08885=1012.138,219.961,-137.263,-53.600,85.418,-53.948
C08886=1012.135,219.688,-137.232,-53.520,85.409,-53.865
C08887=1012.133,219.407,-137.201,-53.433,85.399,-53.775
C08888=1012.129,219.111,-137.169,-53.346,85.389,-53.685
C08889=1012.126,218.807,-137.135,-53.260,85.379,-53.596
C08890=1012.124,218.511,-137.102,-53.174,85.370,-53.506
C08891=1012.121,218.218,-137.069,-53.088,85.360,-53.418
C08892=1012.118,217.928,-137.038,-53.003,85.350,-53.329
C08893=1012.115,217.648,-137.007,-52.925,85.340,-53.249
C08894=1012.112,217.384,-136.977,-52.848,85.331,-53.169
C08895=1012.111,217.123,-136.948,-52.778,85.322,-53.098
C08896=1012.108,216.869,-136.920,-52.708,85.313,-53.026
C08897=1012.106,216.620,-136.893,-52.639,85.304,-52.955
C08898=1012.104,216.375,-136.866,-52.570,85.295,-52.884
C08899=1012.101,216.129,-136.839,-52.502,85.287,-52.814
C08900=1012.099,215.883,-136.812,-52.433,85.278,-52.744
C08901=1012.096,215.638,-136.785,-52.366,85.270,-52.674
C08902=1012.094,215.392,-136.758,-52.298,85.261,-52.604
C08903=1012.093,215.147,-136.731,-52.231,85.253,-52.534
C08904=1012.089,214.903,-136.704,-52.164,85.243,-52.465
C08905=1012.087,214.657,-136.677,-52.097,85.235,-52.396
C08906=1012.086,214.412,-136.650,-52.030,85.226,-52.327
C08907=1012.083,214.168,-136.623,-51.964,85.218,-52.259
C08908=1012.081,213.924,-136.596,-51.898,85.209,-52.191
C08909=1012.079,213.680,-136.569,-51.832,85.200,-52.123
C08910=1012.077,213.436,-136.542,-51.766,85.192,-52.055
C08911=1012.074,213.191,-136.516,-51.701,85.183,-51.987
C08912=1012.072,212.947,-136.489,-51.636,85.174,-51.920
C08913=1012.070,212.704,-136.463,-51.571,85.165,-51.853
C08914=1012.068,212.461,-136.436,-51.506,85.157,-51.786
C08915=1012.065,212.217,-136.408,-51.442,85.148,-51.720
C08916=1012.063,211.974,-136.381,-51.377,85.139,-51.653
C08917=1012.061,211.731,-136.355,-51.314,85.131,-51.587
